// ---- VISUs/Keypad.TcVIS
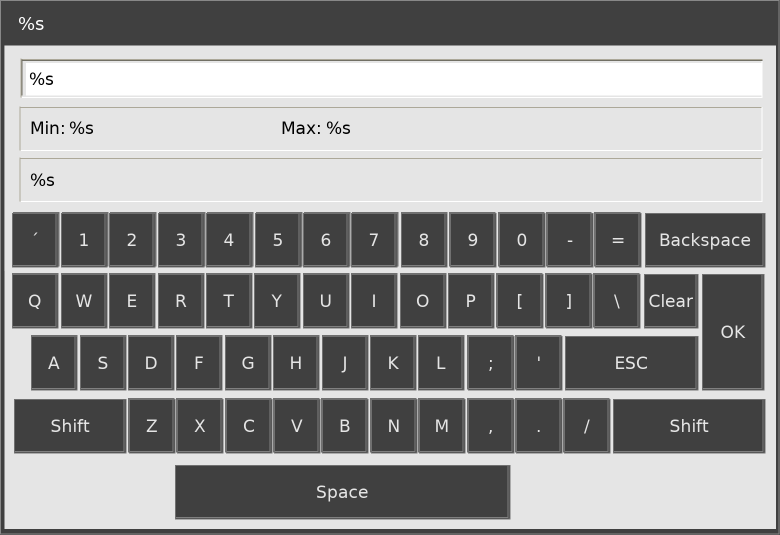
VISUALIZATION Keypad  // 780x535
VAR_INPUT
	stVariableValue : STRING;
	stMin : STRING;
	stMax : STRING;
	stTitle : STRING;
	flags : DWORD;
END_VAR
VAR
	bInit : BOOL;
	bShift : BOOL;
	stMessage : STRING;
	stOutputValue : STRING;
END_VAR
    Rectangle (5,201 772x70)
    Rectangle (3,271 775x62)
    Rectangle (3,333 775x63)
    Rectangle (3,396 775x62)
    Rectangle (3,455 775x75)
    Button (702,274 62x116), "OK"
        OnMouseDown: CloseDialog Dialog=Keypad, Result=OK, NumpadKeypad=True, NumpadKeypadSet=True
    Button (565,336 133x54), "ESC"
        OnMouseDown: CloseDialog Dialog=Keypad, Result=Cancel, NumpadKeypad=True, NumpadKeypadSet=True
    Button (644,274 54x54), "Clear"
        OnMouseDown: execute { stVariableValue := ''; stOutputValue := ''; }
    Button (645,213 120x54), "Backspace"
        OnMouseDown: execute { VisuDlg_CheckedBack(stOutputValue, stVariableValue, bInit); }
    Button (613,399 152x54), "Shift"
        OnMouseDown: toggle bShift
    Button (175,465 335x54), "Space"
        OnMouseDown: execute { VisuDlg_CheckedAppend(stOutputValue, stVariableValue, bInit, (flags AND VisuElems.Visu_InputFlags.Password) = 1, ' '); }
    Button (593,273 46x54), "|", invisible if: NOT bShift
        OnMouseDown: execute { VisuDlg_CheckedAppend(stOutputValue, stVariableValue, bInit, (flags AND VisuElems.Visu_InputFlags.Password) = 1, '|'); }
    Button (467,398 46x54), "<", invisible if: NOT bShift
        OnMouseDown: execute { VisuDlg_CheckedAppend(stOutputValue, stVariableValue, bInit, (flags AND VisuElems.Visu_InputFlags.Password) = 1, '<'); }
    Button (515,398 46x54), ">", invisible if: NOT bShift
        OnMouseDown: execute { VisuDlg_CheckedAppend(stOutputValue, stVariableValue, bInit, (flags AND VisuElems.Visu_InputFlags.Password) = 1, '>'); }
    Button (254,273 46x54), "y", invisible if: NOT bShift
        OnMouseDown: execute { VisuDlg_CheckedAppend(stOutputValue, stVariableValue, bInit, (flags AND VisuElems.Visu_InputFlags.Password) = 1, 'y'); }
    Button (254,274 46x54), "Y", invisible if: bShift
        OnMouseDown: execute { VisuDlg_CheckedAppend(stOutputValue, stVariableValue, bInit, (flags AND VisuElems.Visu_InputFlags.Password) = 1, 'Y'); }
    Button (176,398 46x54), "x", invisible if: NOT bShift
        OnMouseDown: execute { VisuDlg_CheckedAppend(stOutputValue, stVariableValue, bInit, (flags AND VisuElems.Visu_InputFlags.Password) = 1, 'x'); }
    Button (177,399 46x54), "X", invisible if: bShift
        OnMouseDown: execute { VisuDlg_CheckedAppend(stOutputValue, stVariableValue, bInit, (flags AND VisuElems.Visu_InputFlags.Password) = 1, 'X'); }
    Button (225,398 46x54), "c", invisible if: NOT bShift
        OnMouseDown: execute { VisuDlg_CheckedAppend(stOutputValue, stVariableValue, bInit, (flags AND VisuElems.Visu_InputFlags.Password) = 1, 'c'); }
    Button (226,399 46x54), "C", invisible if: bShift
        OnMouseDown: execute { VisuDlg_CheckedAppend(stOutputValue, stVariableValue, bInit, (flags AND VisuElems.Visu_InputFlags.Password) = 1, 'C'); }
    Button (273,398 46x54), "v", invisible if: NOT bShift
        OnMouseDown: execute { VisuDlg_CheckedAppend(stOutputValue, stVariableValue, bInit, (flags AND VisuElems.Visu_InputFlags.Password) = 1, 'v'); }
    Button (274,399 46x54), "V", invisible if: bShift
        OnMouseDown: execute { VisuDlg_CheckedAppend(stOutputValue, stVariableValue, bInit, (flags AND VisuElems.Visu_InputFlags.Password) = 1, 'V'); }
    Button (321,398 46x54), "b", invisible if: NOT bShift
        OnMouseDown: execute { VisuDlg_CheckedAppend(stOutputValue, stVariableValue, bInit, (flags AND VisuElems.Visu_InputFlags.Password) = 1, 'b'); }
    Button (322,399 46x54), "B", invisible if: bShift
        OnMouseDown: execute { VisuDlg_CheckedAppend(stOutputValue, stVariableValue, bInit, (flags AND VisuElems.Visu_InputFlags.Password) = 1, 'B'); }
    Button (370,398 46x54), "n", invisible if: NOT bShift
        OnMouseDown: execute { VisuDlg_CheckedAppend(stOutputValue, stVariableValue, bInit, (flags AND VisuElems.Visu_InputFlags.Password) = 1, 'n'); }
    Button (371,399 46x54), "N", invisible if: bShift
        OnMouseDown: execute { VisuDlg_CheckedAppend(stOutputValue, stVariableValue, bInit, (flags AND VisuElems.Visu_InputFlags.Password) = 1, 'N'); }
    Button (418,398 46x54), "m", invisible if: NOT bShift
        OnMouseDown: execute { VisuDlg_CheckedAppend(stOutputValue, stVariableValue, bInit, (flags AND VisuElems.Visu_InputFlags.Password) = 1, 'm'); }
    Button (419,399 46x54), "M", invisible if: bShift
        OnMouseDown: execute { VisuDlg_CheckedAppend(stOutputValue, stVariableValue, bInit, (flags AND VisuElems.Visu_InputFlags.Password) = 1, 'M'); }
    Button (467,335 46x54), ":", invisible if: NOT bShift
        OnMouseDown: execute { VisuDlg_CheckedAppend(stOutputValue, stVariableValue, bInit, (flags AND VisuElems.Visu_InputFlags.Password) = 1, ':'); }
    Button (546,212 45x54), "_", invisible if: NOT bShift
        OnMouseDown: execute { VisuDlg_CheckedAppend(stOutputValue, stVariableValue, bInit, (flags AND VisuElems.Visu_InputFlags.Password) = 1, '_'); }
    Button (31,335 46x54), "a", invisible if: NOT bShift
        OnMouseDown: execute { VisuDlg_CheckedAppend(stOutputValue, stVariableValue, bInit, (flags AND VisuElems.Visu_InputFlags.Password) = 1, 'a'); }
    Button (31,336 46x54), "A", invisible if: bShift
        OnMouseDown: execute { VisuDlg_CheckedAppend(stOutputValue, stVariableValue, bInit, (flags AND VisuElems.Visu_InputFlags.Password) = 1, 'A'); }
    Button (80,335 46x54), "s", invisible if: NOT bShift
        OnMouseDown: execute { VisuDlg_CheckedAppend(stOutputValue, stVariableValue, bInit, (flags AND VisuElems.Visu_InputFlags.Password) = 1, 's'); }
    Button (80,336 46x54), "S", invisible if: bShift
        OnMouseDown: execute { VisuDlg_CheckedAppend(stOutputValue, stVariableValue, bInit, (flags AND VisuElems.Visu_InputFlags.Password) = 1, 'S'); }
    Button (128,335 46x54), "d", invisible if: NOT bShift
        OnMouseDown: execute { VisuDlg_CheckedAppend(stOutputValue, stVariableValue, bInit, (flags AND VisuElems.Visu_InputFlags.Password) = 1, 'd'); }
    Button (128,336 46x54), "D", invisible if: bShift
        OnMouseDown: execute { VisuDlg_CheckedAppend(stOutputValue, stVariableValue, bInit, (flags AND VisuElems.Visu_InputFlags.Password) = 1, 'D'); }
    Button (176,335 46x54), "f", invisible if: NOT bShift
        OnMouseDown: execute { VisuDlg_CheckedAppend(stOutputValue, stVariableValue, bInit, (flags AND VisuElems.Visu_InputFlags.Password) = 1, 'f'); }
    Button (176,336 46x54), "F", invisible if: bShift
        OnMouseDown: execute { VisuDlg_CheckedAppend(stOutputValue, stVariableValue, bInit, (flags AND VisuElems.Visu_InputFlags.Password) = 1, 'F'); }
    Button (225,335 46x54), "g", invisible if: NOT bShift
        OnMouseDown: execute { VisuDlg_CheckedAppend(stOutputValue, stVariableValue, bInit, (flags AND VisuElems.Visu_InputFlags.Password) = 1, 'g'); }
    Button (225,336 46x54), "G", invisible if: bShift
        OnMouseDown: execute { VisuDlg_CheckedAppend(stOutputValue, stVariableValue, bInit, (flags AND VisuElems.Visu_InputFlags.Password) = 1, 'G'); }
    Button (273,335 46x54), "h", invisible if: NOT bShift
        OnMouseDown: execute { VisuDlg_CheckedAppend(stOutputValue, stVariableValue, bInit, (flags AND VisuElems.Visu_InputFlags.Password) = 1, 'h'); }
    Button (273,336 46x54), "H", invisible if: bShift
        OnMouseDown: execute { VisuDlg_CheckedAppend(stOutputValue, stVariableValue, bInit, (flags AND VisuElems.Visu_InputFlags.Password) = 1, 'H'); }
    Button (322,335 46x54), "j", invisible if: NOT bShift
        OnMouseDown: execute { VisuDlg_CheckedAppend(stOutputValue, stVariableValue, bInit, (flags AND VisuElems.Visu_InputFlags.Password) = 1, 'j'); }
    Button (322,336 46x54), "J", invisible if: bShift
        OnMouseDown: execute { VisuDlg_CheckedAppend(stOutputValue, stVariableValue, bInit, (flags AND VisuElems.Visu_InputFlags.Password) = 1, 'J'); }
    Button (370,335 46x54), "k", invisible if: NOT bShift
        OnMouseDown: execute { VisuDlg_CheckedAppend(stOutputValue, stVariableValue, bInit, (flags AND VisuElems.Visu_InputFlags.Password) = 1, 'k'); }
    Button (370,336 46x54), "K", invisible if: bShift
        OnMouseDown: execute { VisuDlg_CheckedAppend(stOutputValue, stVariableValue, bInit, (flags AND VisuElems.Visu_InputFlags.Password) = 1, 'K'); }
    Button (418,335 46x54), "l", invisible if: NOT bShift
        OnMouseDown: execute { VisuDlg_CheckedAppend(stOutputValue, stVariableValue, bInit, (flags AND VisuElems.Visu_InputFlags.Password) = 1, 'l'); }
    Button (418,336 46x54), "L", invisible if: bShift
        OnMouseDown: execute { VisuDlg_CheckedAppend(stOutputValue, stVariableValue, bInit, (flags AND VisuElems.Visu_InputFlags.Password) = 1, 'L'); }
    Button (159,212 46x54), "#", invisible if: NOT bShift
        OnMouseDown: execute { VisuDlg_CheckedAppend(stOutputValue, stVariableValue, bInit, (flags AND VisuElems.Visu_InputFlags.Password) = 1, '#'); }
    Button (110,212 46x54), "@", invisible if: NOT bShift
        OnMouseDown: execute { VisuDlg_CheckedAppend(stOutputValue, stVariableValue, bInit, (flags AND VisuElems.Visu_InputFlags.Password) = 1, '@'); }
    Button (12,273 46x54), "q", invisible if: NOT bShift
        OnMouseDown: execute { VisuDlg_CheckedAppend(stOutputValue, stVariableValue, bInit, (flags AND VisuElems.Visu_InputFlags.Password) = 1, 'q'); }
    Button (12,274 46x54), "Q", invisible if: bShift
        OnMouseDown: execute { VisuDlg_CheckedAppend(stOutputValue, stVariableValue, bInit, (flags AND VisuElems.Visu_InputFlags.Password) = 1, 'Q'); }
    Button (61,273 46x54), "w", invisible if: NOT bShift
        OnMouseDown: execute { VisuDlg_CheckedAppend(stOutputValue, stVariableValue, bInit, (flags AND VisuElems.Visu_InputFlags.Password) = 1, 'w'); }
    Button (61,274 46x54), "W", invisible if: bShift
        OnMouseDown: execute { VisuDlg_CheckedAppend(stOutputValue, stVariableValue, bInit, (flags AND VisuElems.Visu_InputFlags.Password) = 1, 'W'); }
    Button (109,273 46x54), "e", invisible if: NOT bShift
        OnMouseDown: execute { VisuDlg_CheckedAppend(stOutputValue, stVariableValue, bInit, (flags AND VisuElems.Visu_InputFlags.Password) = 1, 'e'); }
    Button (109,274 46x54), "E", invisible if: bShift
        OnMouseDown: execute { VisuDlg_CheckedAppend(stOutputValue, stVariableValue, bInit, (flags AND VisuElems.Visu_InputFlags.Password) = 1, 'E'); }
    Button (158,273 46x54), "r", invisible if: NOT bShift
        OnMouseDown: execute { VisuDlg_CheckedAppend(stOutputValue, stVariableValue, bInit, (flags AND VisuElems.Visu_InputFlags.Password) = 1, 'r'); }
    Button (158,274 46x54), "R", invisible if: bShift
        OnMouseDown: execute { VisuDlg_CheckedAppend(stOutputValue, stVariableValue, bInit, (flags AND VisuElems.Visu_InputFlags.Password) = 1, 'R'); }
    Button (206,273 46x54), "t", invisible if: NOT bShift
        OnMouseDown: execute { VisuDlg_CheckedAppend(stOutputValue, stVariableValue, bInit, (flags AND VisuElems.Visu_InputFlags.Password) = 1, 't'); }
    Button (206,274 46x54), "T", invisible if: bShift
        OnMouseDown: execute { VisuDlg_CheckedAppend(stOutputValue, stVariableValue, bInit, (flags AND VisuElems.Visu_InputFlags.Password) = 1, 'T'); }
    Button (128,398 46x54), "z", invisible if: NOT bShift
        OnMouseDown: execute { VisuDlg_CheckedAppend(stOutputValue, stVariableValue, bInit, (flags AND VisuElems.Visu_InputFlags.Password) = 1, 'z'); }
    Button (129,399 46x54), "Z", invisible if: bShift
        OnMouseDown: execute { VisuDlg_CheckedAppend(stOutputValue, stVariableValue, bInit, (flags AND VisuElems.Visu_InputFlags.Password) = 1, 'Z'); }
    Button (303,273 46x54), "u", invisible if: NOT bShift
        OnMouseDown: execute { VisuDlg_CheckedAppend(stOutputValue, stVariableValue, bInit, (flags AND VisuElems.Visu_InputFlags.Password) = 1, 'u'); }
    Button (303,274 46x54), "U", invisible if: bShift
        OnMouseDown: execute { VisuDlg_CheckedAppend(stOutputValue, stVariableValue, bInit, (flags AND VisuElems.Visu_InputFlags.Password) = 1, 'U'); }
    Button (351,273 46x54), "i", invisible if: NOT bShift
        OnMouseDown: execute { VisuDlg_CheckedAppend(stOutputValue, stVariableValue, bInit, (flags AND VisuElems.Visu_InputFlags.Password) = 1, 'i'); }
    Button (351,274 46x54), "I", invisible if: bShift
        OnMouseDown: execute { VisuDlg_CheckedAppend(stOutputValue, stVariableValue, bInit, (flags AND VisuElems.Visu_InputFlags.Password) = 1, 'I'); }
    Button (400,273 46x54), "o", invisible if: NOT bShift
        OnMouseDown: execute { VisuDlg_CheckedAppend(stOutputValue, stVariableValue, bInit, (flags AND VisuElems.Visu_InputFlags.Password) = 1, 'o'); }
    Button (400,274 46x54), "O", invisible if: bShift
        OnMouseDown: execute { VisuDlg_CheckedAppend(stOutputValue, stVariableValue, bInit, (flags AND VisuElems.Visu_InputFlags.Password) = 1, 'O'); }
    Button (448,273 46x54), "p", invisible if: NOT bShift
        OnMouseDown: execute { VisuDlg_CheckedAppend(stOutputValue, stVariableValue, bInit, (flags AND VisuElems.Visu_InputFlags.Password) = 1, 'p'); }
    Button (448,274 46x54), "P", invisible if: bShift
        OnMouseDown: execute { VisuDlg_CheckedAppend(stOutputValue, stVariableValue, bInit, (flags AND VisuElems.Visu_InputFlags.Password) = 1, 'P'); }
    Button (594,212 46x54), "+", invisible if: NOT bShift
        OnMouseDown: execute { VisuDlg_CheckedAppend(stOutputValue, stVariableValue, bInit, (flags AND VisuElems.Visu_InputFlags.Password) = 1, '+'); }
    Button (401,212 46x54), "*", invisible if: NOT bShift
        OnMouseDown: execute { VisuDlg_CheckedAppend(stOutputValue, stVariableValue, bInit, (flags AND VisuElems.Visu_InputFlags.Password) = 1, '*'); }
    Button (13,212 46x54), "~", invisible if: NOT bShift
        OnMouseDown: execute { VisuDlg_CheckedAppend(stOutputValue, stVariableValue, bInit, (flags AND VisuElems.Visu_InputFlags.Password) = 1, '~'); }
    Button (304,212 46x54), "^", invisible if: NOT bShift
        OnMouseDown: execute { VisuDlg_CheckedAppend(stOutputValue, stVariableValue, bInit, (flags AND VisuElems.Visu_InputFlags.Password) = 1, '^'); }
    Button (62,212 46x54), "!", invisible if: NOT bShift
        OnMouseDown: execute { VisuDlg_CheckedAppend(stOutputValue, stVariableValue, bInit, (flags AND VisuElems.Visu_InputFlags.Password) = 1, '!'); }
    Button (515,335 46x54), """, invisible if: NOT bShift
        OnMouseDown: execute { VisuDlg_CheckedAppend(stOutputValue, stVariableValue, bInit, (flags AND VisuElems.Visu_InputFlags.Password) = 1, '"'); }
    Button (207,212 46x54), "$", invisible if: NOT bShift
        OnMouseDown: execute { VisuDlg_CheckedAppend(stOutputValue, stVariableValue, bInit, (flags AND VisuElems.Visu_InputFlags.Password) = 1, '$$'); }
    Button (256,212 46x54), "%", invisible if: NOT bShift
        OnMouseDown: execute { VisuDlg_CheckedAppend(stOutputValue, stVariableValue, bInit, (flags AND VisuElems.Visu_InputFlags.Password) = 1, '%'); }
    Button (352,212 46x54), "&", invisible if: NOT bShift
        OnMouseDown: execute { VisuDlg_CheckedAppend(stOutputValue, stVariableValue, bInit, (flags AND VisuElems.Visu_InputFlags.Password) = 1, '&'); }
    Button (449,212 46x54), "(", invisible if: NOT bShift
        OnMouseDown: execute { VisuDlg_CheckedAppend(stOutputValue, stVariableValue, bInit, (flags AND VisuElems.Visu_InputFlags.Password) = 1, '('); }
    Button (498,212 46x54), ")", invisible if: NOT bShift
        OnMouseDown: execute { VisuDlg_CheckedAppend(stOutputValue, stVariableValue, bInit, (flags AND VisuElems.Visu_InputFlags.Password) = 1, ')'); }
    Button (563,398 46x54), "?", invisible if: NOT bShift
        OnMouseDown: execute { VisuDlg_CheckedAppend(stOutputValue, stVariableValue, bInit, (flags AND VisuElems.Visu_InputFlags.Password) = 1, '?'); }
    Rectangle (5,104 773x97)
    Rectangle (27,164 734x32), "%s", text variable: stMessage
    Rectangle (5,42 773x62)
    Rectangle (776,0 4x530)
    Rectangle (0,2 4x527)
    Rectangle (0,529 780x6)
    Polyline (20,201) (20,158) (762,158)
    Polyline (20,150) (20,107) (762,107)
    Polyline (21,97) (21,59) (762,59)
    Polyline (21,201) (762,201) (762,158)
    Polyline (21,150) (762,150) (762,107)
    Polyline (22,97) (762,97) (762,60)
    Rectangle (0,0 779x45)
    Rectangle (15,8 757x32), "%s", text variable: stTitle
    Polyline (22,95) (22,60) (762,60)
    Rectangle (26,63 736x32), "%s", text variable: stOutputValue
    Rectangle (27,112 42x32), "Min:", text variable: stMin, invisible if: LEN(stMin) = 0
    Rectangle (66,112 157x32), "%s", text variable: stMin, invisible if: LEN(stMin) = 0
    Rectangle (278,112 45x32), "Max:", text variable: stMin, invisible if: LEN(stMax) = 0
    Rectangle (323,112 217x32), "%s", text variable: stMax, invisible if: LEN(stMax) = 0
    Button (12,213 46x54), "´", invisible if: bShift
        OnMouseDown: execute { VisuDlg_CheckedAppend(stOutputValue, stVariableValue, bInit, (flags AND VisuElems.Visu_InputFlags.Password) = 1, '´'); }
    Button (61,213 46x54), "1", invisible if: bShift
        OnMouseDown: execute { VisuDlg_CheckedAppend(stOutputValue, stVariableValue, bInit, (flags AND VisuElems.Visu_InputFlags.Password) = 1, '1'); }
    Button (109,213 46x54), "2", invisible if: bShift
        OnMouseDown: execute { VisuDlg_CheckedAppend(stOutputValue, stVariableValue, bInit, (flags AND VisuElems.Visu_InputFlags.Password) = 1, '2'); }
    Button (158,213 46x54), "3", invisible if: bShift
        OnMouseDown: execute { VisuDlg_CheckedAppend(stOutputValue, stVariableValue, bInit, (flags AND VisuElems.Visu_InputFlags.Password) = 1, '3'); }
    Button (206,213 46x54), "4", invisible if: bShift
        OnMouseDown: execute { VisuDlg_CheckedAppend(stOutputValue, stVariableValue, bInit, (flags AND VisuElems.Visu_InputFlags.Password) = 1, '4'); }
    Button (255,213 46x54), "5", invisible if: bShift
        OnMouseDown: execute { VisuDlg_CheckedAppend(stOutputValue, stVariableValue, bInit, (flags AND VisuElems.Visu_InputFlags.Password) = 1, '5'); }
    Button (303,213 46x54), "6", invisible if: bShift
        OnMouseDown: execute { VisuDlg_CheckedAppend(stOutputValue, stVariableValue, bInit, (flags AND VisuElems.Visu_InputFlags.Password) = 1, '6'); }
    Button (351,213 46x54), "7", invisible if: bShift
        OnMouseDown: execute { VisuDlg_CheckedAppend(stOutputValue, stVariableValue, bInit, (flags AND VisuElems.Visu_InputFlags.Password) = 1, '7'); }
    Button (401,213 46x54), "8", invisible if: bShift
        OnMouseDown: execute { VisuDlg_CheckedAppend(stOutputValue, stVariableValue, bInit, (flags AND VisuElems.Visu_InputFlags.Password) = 1, '8'); }
    Button (450,213 46x54), "9", invisible if: bShift
        OnMouseDown: execute { VisuDlg_CheckedAppend(stOutputValue, stVariableValue, bInit, (flags AND VisuElems.Visu_InputFlags.Password) = 1, '9'); }
    Button (499,213 46x54), "0", invisible if: bShift
        OnMouseDown: execute { VisuDlg_CheckedAppend(stOutputValue, stVariableValue, bInit, (flags AND VisuElems.Visu_InputFlags.Password) = 1, '0'); }
    Button (547,213 46x54), "-", invisible if: bShift
        OnMouseDown: execute { VisuDlg_CheckedAppend(stOutputValue, stVariableValue, bInit, (flags AND VisuElems.Visu_InputFlags.Password) = 1, '-'); }
    Button (595,213 46x54), "=", invisible if: bShift
        OnMouseDown: execute { VisuDlg_CheckedAppend(stOutputValue, stVariableValue, bInit, (flags AND VisuElems.Visu_InputFlags.Password) = 1, '='); }
    Button (496,273 46x54), "{", invisible if: NOT bShift
        OnMouseDown: execute { VisuDlg_CheckedAppend(stOutputValue, stVariableValue, bInit, (flags AND VisuElems.Visu_InputFlags.Password) = 1, '{'); }
    Button (497,274 46x54), "[", invisible if: bShift
        OnMouseDown: execute { VisuDlg_CheckedAppend(stOutputValue, stVariableValue, bInit, (flags AND VisuElems.Visu_InputFlags.Password) = 1, '['); }
    Button (545,273 46x54), "}", invisible if: NOT bShift
        OnMouseDown: execute { VisuDlg_CheckedAppend(stOutputValue, stVariableValue, bInit, (flags AND VisuElems.Visu_InputFlags.Password) = 1, '}'); }
    Button (546,274 46x54), "]", invisible if: bShift
        OnMouseDown: execute { VisuDlg_CheckedAppend(stOutputValue, stVariableValue, bInit, (flags AND VisuElems.Visu_InputFlags.Password) = 1, ']'); }
    Button (594,274 46x54), "\", invisible if: bShift
        OnMouseDown: execute { VisuDlg_CheckedAppend(stOutputValue, stVariableValue, bInit, (flags AND VisuElems.Visu_InputFlags.Password) = 1, '\'); }
    Button (468,336 46x54), ";", invisible if: bShift
        OnMouseDown: execute { VisuDlg_CheckedAppend(stOutputValue, stVariableValue, bInit, (flags AND VisuElems.Visu_InputFlags.Password) = 1, ';'); }
    Button (516,336 46x54), "'", invisible if: bShift
        OnMouseDown: execute { VisuDlg_CheckedAppend(stOutputValue, stVariableValue, bInit, (flags AND VisuElems.Visu_InputFlags.Password) = 1, '$''); }
    Button (468,399 46x54), ",", invisible if: bShift
        OnMouseDown: execute { VisuDlg_CheckedAppend(stOutputValue, stVariableValue, bInit, (flags AND VisuElems.Visu_InputFlags.Password) = 1, ','); }
    Button (516,399 46x54), ".", invisible if: bShift
        OnMouseDown: execute { VisuDlg_CheckedAppend(stOutputValue, stVariableValue, bInit, (flags AND VisuElems.Visu_InputFlags.Password) = 1, '.'); }
    Button (564,399 46x54), "/", invisible if: bShift
        OnMouseDown: execute { VisuDlg_CheckedAppend(stOutputValue, stVariableValue, bInit, (flags AND VisuElems.Visu_InputFlags.Password) = 1, '/'); }
    Button (14,399 112x54), "Shift"
        OnMouseDown: toggle bShift
    hotkey HotkeyInput Id=481083523072, Key=KeyDown=True, KeyName=BACKSPACE, ActionToExecute=Action=STSnippet=VisuDlg_CheckedBack(stOutputValue, stVariableValue, bInit);, VisuElemId=-1
    hotkey HotkeyInput Id=481084571648, Key=KeyDown=True, KeyName=DELETE, ActionToExecute=Action=STSnippet=stVariableValue := ''; stOutputValue := '';, VisuElemId=-1
    hotkey HotkeyInput Id=481085620224, Key=KeyDown=True, KeyName=ESCAPE, ActionToExecute=Action=Dialog=Keypad, Result=Cancel, NumpadKeypad=True, NumpadKeypadSet=True, VisuElemId=-1
    hotkey HotkeyInput Id=481086668800, Key=KeyDown=True, KeyName=SPACE, ActionToExecute=Action=STSnippet=VisuDlg_CheckedAppend(stOutputValue, stVariableValue, bInit, (flags AND VisuElems.Visu_InputFlags.Password) = 1, ' ');, VisuElemId=-1
    hotkey HotkeyInput Id=481087717376, Key=Modifiers=1, KeyDown=True, KeyName=SPACE, ActionToExecute=Action=ToggleVariable=bShift, VisuElemId=-1
    hotkey HotkeyInput Id=481088765952, Key=KeyDown=True, KeyName=RETURN_KEY, ActionToExecute=Action=Dialog=Keypad, Result=OK, NumpadKeypad=True, NumpadKeypadSet=True, VisuElemId=-1
    hotkey HotkeyInput Id=481089814528, Key=KeyDown=True, KeyName=1, ActionToExecute=Action=STSnippet=IF bShift THEN VisuDlg_CheckedAppend(stOutputValue, stVariableValue, bInit, (flags AND VisuElems.Visu_InputFlags.Password) = 1, '!'); ELSE VisuDlg_CheckedAppend(stOutputValue, stVariableValue, bInit, (flags AND VisuElems.Visu_InputFlags.Password) = 1, '1'); END_IF, VisuElemId=-1
    hotkey HotkeyInput Id=481090863104, Key=KeyDown=True, KeyName=2, ActionToExecute=Action=STSnippet=IF bShift THEN VisuDlg_CheckedAppend(stOutputValue, stVariableValue, bInit, (flags AND VisuElems.Visu_InputFlags.Password) = 1, '@'); ELSE VisuDlg_CheckedAppend(stOutputValue, stVariableValue, bInit, (flags AND VisuElems.Visu_InputFlags.Password) = 1, '2'); END_IF, VisuElemId=-1
    hotkey HotkeyInput Id=481091911680, Key=KeyDown=True, KeyName=3, ActionToExecute=Action=STSnippet=IF bShift THEN VisuDlg_CheckedAppend(stOutputValue, stVariableValue, bInit, (flags AND VisuElems.Visu_InputFlags.Password) = 1, '#'); ELSE VisuDlg_CheckedAppend(stOutputValue, stVariableValue, bInit, (flags AND VisuElems.Visu_InputFlags.Password) = 1, '3'); END_IF, VisuElemId=-1
    hotkey HotkeyInput Id=481092960256, Key=KeyDown=True, KeyName=4, ActionToExecute=Action=STSnippet=IF bShift THEN VisuDlg_CheckedAppend(stOutputValue, stVariableValue, bInit, (flags AND VisuElems.Visu_InputFlags.Password) = 1, '$$'); ELSE VisuDlg_CheckedAppend(stOutputValue, stVariableValue, bInit, (flags AND VisuElems.Visu_InputFlags.Password) = 1, '4'); END_IF, VisuElemId=-1
    hotkey HotkeyInput Id=481094008832, Key=KeyDown=True, KeyName=5, ActionToExecute=Action=STSnippet=IF bShift THEN VisuDlg_CheckedAppend(stOutputValue, stVariableValue, bInit, (flags AND VisuElems.Visu_InputFlags.Password) = 1, '%'); ELSE VisuDlg_CheckedAppend(stOutputValue, stVariableValue, bInit, (flags AND VisuElems.Visu_InputFlags.Password) = 1, '5'); END_IF, VisuElemId=-1
    hotkey HotkeyInput Id=481095057408, Key=KeyDown=True, KeyName=6, ActionToExecute=Action=STSnippet=IF bShift THEN VisuDlg_CheckedAppend(stOutputValue, stVariableValue, bInit, (flags AND VisuElems.Visu_InputFlags.Password) = 1, '^'); ELSE VisuDlg_CheckedAppend(stOutputValue, stVariableValue, bInit, (flags AND VisuElems.Visu_InputFlags.Password) = 1, '6'); END_IF, VisuElemId=-1
    hotkey HotkeyInput Id=481096105984, Key=KeyDown=True, KeyName=7, ActionToExecute=Action=STSnippet=IF bShift THEN VisuDlg_CheckedAppend(stOutputValue, stVariableValue, bInit, (flags AND VisuElems.Visu_InputFlags.Password) = 1, '&'); ELSE VisuDlg_CheckedAppend(stOutputValue, stVariableValue, bInit, (flags AND VisuElems.Visu_InputFlags.Password) = 1, '7'); END_IF, VisuElemId=-1
    hotkey HotkeyInput Id=481097154560, Key=KeyDown=True, KeyName=8, ActionToExecute=Action=STSnippet=IF bShift THEN VisuDlg_CheckedAppend(stOutputValue, stVariableValue, bInit, (flags AND VisuElems.Visu_InputFlags.Password) = 1, '*'); ELSE VisuDlg_CheckedAppend(stOutputValue, stVariableValue, bInit, (flags AND VisuElems.Visu_InputFlags.Password) = 1, '8'); END_IF, VisuElemId=-1
    hotkey HotkeyInput Id=481098203136, Key=KeyDown=True, KeyName=9, ActionToExecute=Action=STSnippet=IF bShift THEN VisuDlg_CheckedAppend(stOutputValue, stVariableValue, bInit, (flags AND VisuElems.Visu_InputFlags.Password) = 1, '('); ELSE VisuDlg_CheckedAppend(stOutputValue, stVariableValue, bInit, (flags AND VisuElems.Visu_InputFlags.Password) = 1, '9'); END_IF, VisuElemId=-1
    hotkey HotkeyInput Id=481099251712, Key=KeyDown=True, KeyName=0, ActionToExecute=Action=STSnippet=IF bShift THEN VisuDlg_CheckedAppend(stOutputValue, stVariableValue, bInit, (flags AND VisuElems.Visu_InputFlags.Password) = 1, ')'); ELSE VisuDlg_CheckedAppend(stOutputValue, stVariableValue, bInit, (flags AND VisuElems.Visu_InputFlags.Password) = 1, '0'); END_IF, VisuElemId=-1
    hotkey HotkeyInput Id=481100300288, Key=KeyDown=True, KeyName=SUBTRACT, ActionToExecute=Action=STSnippet=IF bShift THEN VisuDlg_CheckedAppend(stOutputValue, stVariableValue, bInit, (flags AND VisuElems.Visu_InputFlags.Password) = 1, '_'); ELSE VisuDlg_CheckedAppend(stOutputValue, stVariableValue, bInit, (flags AND VisuElems.Visu_InputFlags.Password) = 1, '-'); END_IF, VisuElemId=-1
    hotkey HotkeyInput Id=481101348864, Key=KeyDown=True, KeyName=ADDITION, ActionToExecute=Action=STSnippet=IF bShift THEN VisuDlg_CheckedAppend(stOutputValue, stVariableValue, bInit, (flags AND VisuElems.Visu_InputFlags.Password) = 1, '='); ELSE VisuDlg_CheckedAppend(stOutputValue, stVariableValue, bInit, (flags AND VisuElems.Visu_InputFlags.Password) = 1, '+'); END_IF, VisuElemId=-1
    hotkey HotkeyInput Id=481102397440, Key=KeyDown=True, KeyName=Q, ActionToExecute=Action=STSnippet=IF bShift THEN VisuDlg_CheckedAppend(stOutputValue, stVariableValue, bInit, (flags AND VisuElems.Visu_InputFlags.Password) = 1, 'q'); ELSE VisuDlg_CheckedAppend(stOutputValue, stVariableValue, bInit, (flags AND VisuElems.Visu_InputFlags.Password) = 1, 'Q'); END_IF, VisuElemId=-1
    hotkey HotkeyInput Id=481103446016, Key=KeyDown=True, KeyName=W, ActionToExecute=Action=STSnippet=IF bShift THEN VisuDlg_CheckedAppend(stOutputValue, stVariableValue, bInit, (flags AND VisuElems.Visu_InputFlags.Password) = 1, 'w'); ELSE VisuDlg_CheckedAppend(stOutputValue, stVariableValue, bInit, (flags AND VisuElems.Visu_InputFlags.Password) = 1, 'W'); END_IF, VisuElemId=-1
    hotkey HotkeyInput Id=481104494592, Key=KeyDown=True, KeyName=E, ActionToExecute=Action=STSnippet=IF bShift THEN VisuDlg_CheckedAppend(stOutputValue, stVariableValue, bInit, (flags AND VisuElems.Visu_InputFlags.Password) = 1, 'e'); ELSE VisuDlg_CheckedAppend(stOutputValue, stVariableValue, bInit, (flags AND VisuElems.Visu_InputFlags.Password) = 1, 'E'); END_IF, VisuElemId=-1
    hotkey HotkeyInput Id=481105543168, Key=KeyDown=True, KeyName=R, ActionToExecute=Action=STSnippet=IF bShift THEN VisuDlg_CheckedAppend(stOutputValue, stVariableValue, bInit, (flags AND VisuElems.Visu_InputFlags.Password) = 1, 'r'); ELSE VisuDlg_CheckedAppend(stOutputValue, stVariableValue, bInit, (flags AND VisuElems.Visu_InputFlags.Password) = 1, 'R'); END_IF, VisuElemId=-1
    hotkey HotkeyInput Id=481106591744, Key=KeyDown=True, KeyName=T, ActionToExecute=Action=STSnippet=IF bShift THEN VisuDlg_CheckedAppend(stOutputValue, stVariableValue, bInit, (flags AND VisuElems.Visu_InputFlags.Password) = 1, 't'); ELSE VisuDlg_CheckedAppend(stOutputValue, stVariableValue, bInit, (flags AND VisuElems.Visu_InputFlags.Password) = 1, 'T'); END_IF, VisuElemId=-1
    hotkey HotkeyInput Id=481107640320, Key=KeyDown=True, KeyName=Y, ActionToExecute=Action=STSnippet=IF bShift THEN VisuDlg_CheckedAppend(stOutputValue, stVariableValue, bInit, (flags AND VisuElems.Visu_InputFlags.Password) = 1, 'y'); ELSE VisuDlg_CheckedAppend(stOutputValue, stVariableValue, bInit, (flags AND VisuElems.Visu_InputFlags.Password) = 1, 'Y'); END_IF, VisuElemId=-1
    hotkey HotkeyInput Id=481108688896, Key=KeyDown=True, KeyName=U, ActionToExecute=Action=STSnippet=IF bShift THEN VisuDlg_CheckedAppend(stOutputValue, stVariableValue, bInit, (flags AND VisuElems.Visu_InputFlags.Password) = 1, 'u'); ELSE VisuDlg_CheckedAppend(stOutputValue, stVariableValue, bInit, (flags AND VisuElems.Visu_InputFlags.Password) = 1, 'U'); END_IF, VisuElemId=-1
    hotkey HotkeyInput Id=481109737472, Key=KeyDown=True, KeyName=I, ActionToExecute=Action=STSnippet=IF bShift THEN VisuDlg_CheckedAppend(stOutputValue, stVariableValue, bInit, (flags AND VisuElems.Visu_InputFlags.Password) = 1, 'i'); ELSE VisuDlg_CheckedAppend(stOutputValue, stVariableValue, bInit, (flags AND VisuElems.Visu_InputFlags.Password) = 1, 'I'); END_IF, VisuElemId=-1
    hotkey HotkeyInput Id=481110786048, Key=KeyDown=True, KeyName=O, ActionToExecute=Action=STSnippet=IF bShift THEN VisuDlg_CheckedAppend(stOutputValue, stVariableValue, bInit, (flags AND VisuElems.Visu_InputFlags.Password) = 1, 'o'); ELSE VisuDlg_CheckedAppend(stOutputValue, stVariableValue, bInit, (flags AND VisuElems.Visu_InputFlags.Password) = 1, 'O'); END_IF, VisuElemId=-1
    hotkey HotkeyInput Id=481111834624, Key=KeyDown=True, KeyName=P, ActionToExecute=Action=STSnippet=IF bShift THEN VisuDlg_CheckedAppend(stOutputValue, stVariableValue, bInit, (flags AND VisuElems.Visu_InputFlags.Password) = 1, 'p'); ELSE VisuDlg_CheckedAppend(stOutputValue, stVariableValue, bInit, (flags AND VisuElems.Visu_InputFlags.Password) = 1, 'P'); END_IF, VisuElemId=-1
    hotkey HotkeyInput Id=481112883200, Key=KeyDown=True, KeyName=A, ActionToExecute=Action=STSnippet=IF bShift THEN VisuDlg_CheckedAppend(stOutputValue, stVariableValue, bInit, (flags AND VisuElems.Visu_InputFlags.Password) = 1, 'a'); ELSE VisuDlg_CheckedAppend(stOutputValue, stVariableValue, bInit, (flags AND VisuElems.Visu_InputFlags.Password) = 1, 'A'); END_IF, VisuElemId=-1
    hotkey HotkeyInput Id=481113931776, Key=KeyDown=True, KeyName=S, ActionToExecute=Action=STSnippet=IF bShift THEN VisuDlg_CheckedAppend(stOutputValue, stVariableValue, bInit, (flags AND VisuElems.Visu_InputFlags.Password) = 1, 's'); ELSE VisuDlg_CheckedAppend(stOutputValue, stVariableValue, bInit, (flags AND VisuElems.Visu_InputFlags.Password) = 1, 'S'); END_IF, VisuElemId=-1
    hotkey HotkeyInput Id=481114980352, Key=KeyDown=True, KeyName=D, ActionToExecute=Action=STSnippet=IF bShift THEN VisuDlg_CheckedAppend(stOutputValue, stVariableValue, bInit, (flags AND VisuElems.Visu_InputFlags.Password) = 1, 'd'); ELSE VisuDlg_CheckedAppend(stOutputValue, stVariableValue, bInit, (flags AND VisuElems.Visu_InputFlags.Password) = 1, 'D'); END_IF, VisuElemId=-1
    hotkey HotkeyInput Id=481116028928, Key=KeyDown=True, KeyName=F, ActionToExecute=Action=STSnippet=IF bShift THEN VisuDlg_CheckedAppend(stOutputValue, stVariableValue, bInit, (flags AND VisuElems.Visu_InputFlags.Password) = 1, 'f'); ELSE VisuDlg_CheckedAppend(stOutputValue, stVariableValue, bInit, (flags AND VisuElems.Visu_InputFlags.Password) = 1, 'F'); END_IF, VisuElemId=-1
    hotkey HotkeyInput Id=481117077504, Key=KeyDown=True, KeyName=G, ActionToExecute=Action=STSnippet=IF bShift THEN VisuDlg_CheckedAppend(stOutputValue, stVariableValue, bInit, (flags AND VisuElems.Visu_InputFlags.Password) = 1, 'g'); ELSE VisuDlg_CheckedAppend(stOutputValue, stVariableValue, bInit, (flags AND VisuElems.Visu_InputFlags.Password) = 1, 'G'); END_IF, VisuElemId=-1
    hotkey HotkeyInput Id=481118126080, Key=KeyDown=True, KeyName=H, ActionToExecute=Action=STSnippet=IF bShift THEN VisuDlg_CheckedAppend(stOutputValue, stVariableValue, bInit, (flags AND VisuElems.Visu_InputFlags.Password) = 1, 'h'); ELSE VisuDlg_CheckedAppend(stOutputValue, stVariableValue, bInit, (flags AND VisuElems.Visu_InputFlags.Password) = 1, 'H'); END_IF, VisuElemId=-1
    hotkey HotkeyInput Id=481119174656, Key=KeyDown=True, KeyName=J, ActionToExecute=Action=STSnippet=IF bShift THEN VisuDlg_CheckedAppend(stOutputValue, stVariableValue, bInit, (flags AND VisuElems.Visu_InputFlags.Password) = 1, 'j'); ELSE VisuDlg_CheckedAppend(stOutputValue, stVariableValue, bInit, (flags AND VisuElems.Visu_InputFlags.Password) = 1, 'J'); END_IF, VisuElemId=-1
    hotkey HotkeyInput Id=481120223232, Key=KeyDown=True, KeyName=K, ActionToExecute=Action=STSnippet=IF bShift THEN VisuDlg_CheckedAppend(stOutputValue, stVariableValue, bInit, (flags AND VisuElems.Visu_InputFlags.Password) = 1, 'k'); ELSE VisuDlg_CheckedAppend(stOutputValue, stVariableValue, bInit, (flags AND VisuElems.Visu_InputFlags.Password) = 1, 'K'); END_IF, VisuElemId=-1
    hotkey HotkeyInput Id=481121271808, Key=KeyDown=True, KeyName=L, ActionToExecute=Action=STSnippet=IF bShift THEN VisuDlg_CheckedAppend(stOutputValue, stVariableValue, bInit, (flags AND VisuElems.Visu_InputFlags.Password) = 1, 'l'); ELSE VisuDlg_CheckedAppend(stOutputValue, stVariableValue, bInit, (flags AND VisuElems.Visu_InputFlags.Password) = 1, 'L'); END_IF, VisuElemId=-1
    hotkey HotkeyInput Id=481122320384, Key=KeyDown=True, KeyName=Z, ActionToExecute=Action=STSnippet=IF bShift THEN VisuDlg_CheckedAppend(stOutputValue, stVariableValue, bInit, (flags AND VisuElems.Visu_InputFlags.Password) = 1, 'z'); ELSE VisuDlg_CheckedAppend(stOutputValue, stVariableValue, bInit, (flags AND VisuElems.Visu_InputFlags.Password) = 1, 'Z'); END_IF, VisuElemId=-1
    hotkey HotkeyInput Id=481123368960, Key=KeyDown=True, KeyName=X, ActionToExecute=Action=STSnippet=IF bShift THEN VisuDlg_CheckedAppend(stOutputValue, stVariableValue, bInit, (flags AND VisuElems.Visu_InputFlags.Password) = 1, 'x'); ELSE VisuDlg_CheckedAppend(stOutputValue, stVariableValue, bInit, (flags AND VisuElems.Visu_InputFlags.Password) = 1, 'X'); END_IF, VisuElemId=-1
    hotkey HotkeyInput Id=481124417536, Key=KeyDown=True, KeyName=C, ActionToExecute=Action=STSnippet=IF bShift THEN VisuDlg_CheckedAppend(stOutputValue, stVariableValue, bInit, (flags AND VisuElems.Visu_InputFlags.Password) = 1, 'c'); ELSE VisuDlg_CheckedAppend(stOutputValue, stVariableValue, bInit, (flags AND VisuElems.Visu_InputFlags.Password) = 1, 'C'); END_IF, VisuElemId=-1
    hotkey HotkeyInput Id=481125466112, Key=KeyDown=True, KeyName=V, ActionToExecute=Action=STSnippet=IF bShift THEN VisuDlg_CheckedAppend(stOutputValue, stVariableValue, bInit, (flags AND VisuElems.Visu_InputFlags.Password) = 1, 'v'); ELSE VisuDlg_CheckedAppend(stOutputValue, stVariableValue, bInit, (flags AND VisuElems.Visu_InputFlags.Password) = 1, 'V'); END_IF, VisuElemId=-1
    hotkey HotkeyInput Id=481126514688, Key=KeyDown=True, KeyName=B, ActionToExecute=Action=STSnippet=IF bShift THEN VisuDlg_CheckedAppend(stOutputValue, stVariableValue, bInit, (flags AND VisuElems.Visu_InputFlags.Password) = 1, 'b'); ELSE VisuDlg_CheckedAppend(stOutputValue, stVariableValue, bInit, (flags AND VisuElems.Visu_InputFlags.Password) = 1, 'B'); END_IF, VisuElemId=-1
    hotkey HotkeyInput Id=481127563264, Key=KeyDown=True, KeyName=N, ActionToExecute=Action=STSnippet=IF bShift THEN VisuDlg_CheckedAppend(stOutputValue, stVariableValue, bInit, (flags AND VisuElems.Visu_InputFlags.Password) = 1, 'n'); ELSE VisuDlg_CheckedAppend(stOutputValue, stVariableValue, bInit, (flags AND VisuElems.Visu_InputFlags.Password) = 1, 'N'); END_IF, VisuElemId=-1
    hotkey HotkeyInput Id=481128611840, Key=KeyDown=True, KeyName=M, ActionToExecute=Action=STSnippet=IF bShift THEN VisuDlg_CheckedAppend(stOutputValue, stVariableValue, bInit, (flags AND VisuElems.Visu_InputFlags.Password) = 1, 'm'); ELSE VisuDlg_CheckedAppend(stOutputValue, stVariableValue, bInit, (flags AND VisuElems.Visu_InputFlags.Password) = 1, 'M'); END_IF, VisuElemId=-1
    hotkey HotkeyInput Id=481129660416, Key=KeyDown=True, KeyName=COMMA, ActionToExecute=Action=STSnippet=IF bShift THEN VisuDlg_CheckedAppend(stOutputValue, stVariableValue, bInit, (flags AND VisuElems.Visu_InputFlags.Password) = 1, ','); ELSE VisuDlg_CheckedAppend(stOutputValue, stVariableValue, bInit, (flags AND VisuElems.Visu_InputFlags.Password) = 1, '.'); END_IF, VisuElemId=-1
    hotkey HotkeyInput Id=481131757568, Key=KeyDown=True, KeyName=NUM1, ActionToExecute=Action=STSnippet=VisuDlg_CheckedAppend(stOutputValue, stVariableValue, bInit, (flags AND VisuElems.Visu_InputFlags.Password) = 1, '1');, VisuElemId=-1
    hotkey HotkeyInput Id=481132806144, Key=KeyDown=True, KeyName=NUM2, ActionToExecute=Action=STSnippet=VisuDlg_CheckedAppend(stOutputValue, stVariableValue, bInit, (flags AND VisuElems.Visu_InputFlags.Password) = 1, '2');, VisuElemId=-1
    hotkey HotkeyInput Id=481133854720, Key=KeyDown=True, KeyName=NUM3, ActionToExecute=Action=STSnippet=VisuDlg_CheckedAppend(stOutputValue, stVariableValue, bInit, (flags AND VisuElems.Visu_InputFlags.Password) = 1, '3');, VisuElemId=-1
    hotkey HotkeyInput Id=481134903296, Key=KeyDown=True, KeyName=NUM4, ActionToExecute=Action=STSnippet=VisuDlg_CheckedAppend(stOutputValue, stVariableValue, bInit, (flags AND VisuElems.Visu_InputFlags.Password) = 1, '4');, VisuElemId=-1
    hotkey HotkeyInput Id=481135951872, Key=KeyDown=True, KeyName=NUM5, ActionToExecute=Action=STSnippet=VisuDlg_CheckedAppend(stOutputValue, stVariableValue, bInit, (flags AND VisuElems.Visu_InputFlags.Password) = 1, '5');, VisuElemId=-1
    hotkey HotkeyInput Id=481137000448, Key=KeyDown=True, KeyName=NUM6, ActionToExecute=Action=STSnippet=VisuDlg_CheckedAppend(stOutputValue, stVariableValue, bInit, (flags AND VisuElems.Visu_InputFlags.Password) = 1, '6');, VisuElemId=-1
    hotkey HotkeyInput Id=481138049024, Key=KeyDown=True, KeyName=NUM7, ActionToExecute=Action=STSnippet=VisuDlg_CheckedAppend(stOutputValue, stVariableValue, bInit, (flags AND VisuElems.Visu_InputFlags.Password) = 1, '7');, VisuElemId=-1
    hotkey HotkeyInput Id=481139097600, Key=KeyDown=True, KeyName=NUM8, ActionToExecute=Action=STSnippet=VisuDlg_CheckedAppend(stOutputValue, stVariableValue, bInit, (flags AND VisuElems.Visu_InputFlags.Password) = 1, '8');, VisuElemId=-1
    hotkey HotkeyInput Id=481140146176, Key=KeyDown=True, KeyName=NUM9, ActionToExecute=Action=STSnippet=VisuDlg_CheckedAppend(stOutputValue, stVariableValue, bInit, (flags AND VisuElems.Visu_InputFlags.Password) = 1, '9');, VisuElemId=-1
    hotkey HotkeyInput Id=481141194752, Key=KeyDown=True, KeyName=NUM0, ActionToExecute=Action=STSnippet=VisuDlg_CheckedAppend(stOutputValue, stVariableValue, bInit, (flags AND VisuElems.Visu_InputFlags.Password) = 1, '0');, VisuElemId=-1
END_VISUALIZATION

// ---- VISUs/Kierwonica.TcVIS
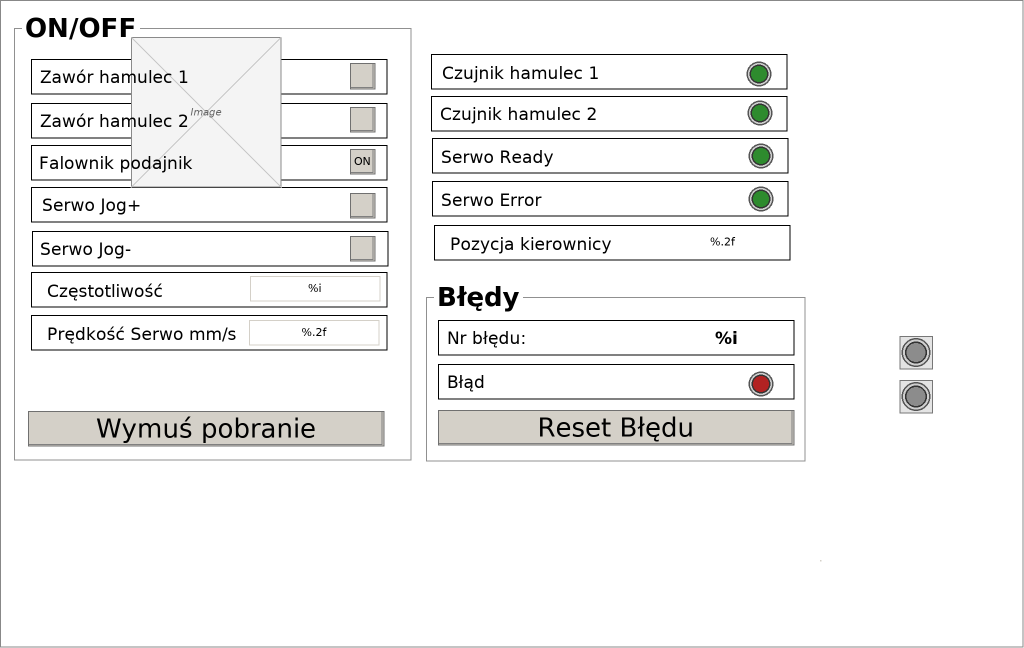
VISUALIZATION Kierwonica  // 1024x648
    Rectangle (31,59 356x35)
    Rectangle (31,103 356x35)
    Rectangle (31,145 356x35)
    Rectangle (31,272 356x35)
    Rectangle (32,231 356x35)
    Rectangle (31,187 356x35)
    GroupBox (14,20 397x440), "ON/OFF"
        Rectangle (17,295 356x35)
        Button (336,173 25x25)
            tap GVL_HMI.bHmiJogF
        Button (336,216 25x25)
            tap GVL_HMI.bHmiJogB
        Textfield (236,256 130x25), "%i", text variable: GVL_HMI.iFreqKierownicaMan
            OnMouseClick: write the text variable via Edit
        Button (336,129 25x25), "ON", colour toggle: GVL_GLOBAL.falownik_podajnik_kier_cewka
            tap GVL_HMI.przycisk_falownik_podajnik_kier
        Button (336,87 25x25), colour toggle: GVL_GLOBAL.zaw_ham2_kier_cewka
            tap GVL_HMI.przycisk_zaw_ham2_kier
        Button (336,43 25x26), colour toggle: GVL_GLOBAL.zaw_ham1_kier_cewka
            tap GVL_HMI.przycisk_zaw_ham1_kier
        Image (117,17 150x150)
        Button (14,391 356x35), "Wymuś pobranie"
            OnMouseDown: execute { GVL_HMI.Wymus_pobranie:=TRUE; }
    Rectangle (431,54 356x35)
    Label (437,57 230x30)
    Rectangle (431,96 356x35)
    Label (437,99 239x30), "Czujnik hamulec 2"
    Lamp1 (746,99 28x28), variable: GVL_IO_K.b4B6, style: Lamp-Lamp1-Green
    Lamp1 (745,60 28x28), variable: GVL_IO_K.b4B7, style: Lamp-Lamp1-Green
    Label (439,58 239x30), "Czujnik hamulec 1"
    Rectangle (432,138 356x35)
    Rectangle (432,181 356x35)
    Label (37,101 239x30)
    Label (37,106 209x30), "Zawór hamulec 2"
    Label (37,62 209x30), "Zawór hamulec 1"
    Label (36,148 209x30), "Falownik podajnik"
    Label (44,276 209x30), "Częstotliwość"
    Label (438,142 239x30), "Serwo Ready"
    Lamp1 (747,142 28x28), variable: PRG_Kierownica.S_K_Power.Status, style: Lamp-Lamp1-Green
    Label (438,185 239x30), "Serwo Error"
    Lamp1 (747,185 28x28), variable: PRG_Kierownica.S_K_Power.Error, style: Lamp-Lamp1-Green
    Rectangle (434,225 356x35)
    Label (447,229 209x30), "Pozycja kierownicy"
    Textfield (662,227 121x30), "%.2f", text variable: GVL_AXIS.stAxis2.NcToPlc.ActPos
    Label (39,190 209x30), "Serwo Jog+"
    Label (37,234 209x30), "Serwo Jog-"
    PushSwitch (897,380 38x33), behaviour: TOGGLE, style: Switch-PushSwitch-Gray
    PushSwitch (897,336 38x33), behaviour: TOGGLE, style: Switch-PushSwitch-Gray
    Textfield (249,320 130x25), "%.2f", text variable: gvl_hmi.J_Vel
        OnMouseClick: write the text variable via Edit
    Label (44,319 209x30), "Prędkość Serwo mm/s"
    Textfield (820,560 1x1)
    GroupBox (426,289 379x172), "Błędy"
        Rectangle (12,31 356x35)
        Label (18,34 209x30), "Nr błędu:"
        Rectangle (12,75 356x35)
        Label (18,78 209x30), "Błąd"
        Button (12,121 356x35), "Reset Błędu"
            tap GVL_HMI.ErrorResetKier
        Lamp1 (321,81 28x28), variable: GVL_GLOBAL.Error_pakowania, style: Lamp-Lamp1-Red
        Textfield (240,34 121x30), "%i", text variable: GVL_GLOBAL.Error_numb_kier
END_VISUALIZATION

// ---- VISUs/mssgbox.TcVIS
VISUALIZATION mssgbox  // 200x100
END_VISUALIZATION

// ---- VISUs/PH_AxisOnline.TcVIS
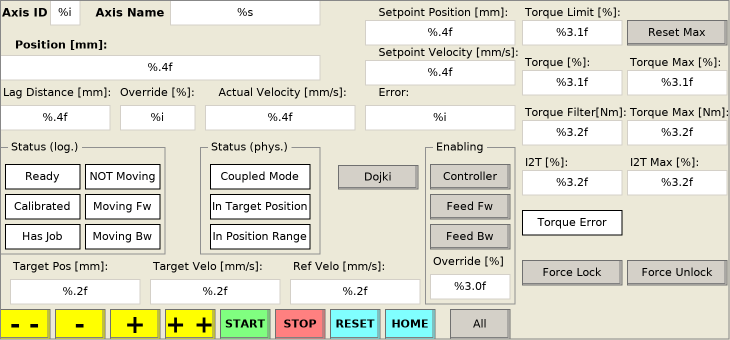
VISUALIZATION PH_AxisOnline  // 730x340
//==================================================================================================
//							Beckhoff Automation Poland
//									18.04.2018
//	Wizualizacja dla Axis Online
//  v1.0	|| TC v 3.1.4022.16		|| - pierwsza wersja
//==================================================================================================
VAR_IN_OUT
	stMcAxisOnline			: ST_McAxisOnline;	
END_VAR
    Frame (0,0 520x340)
        shows PH_NcAxis(stMcAxisOnline := stMcAxisOnline)
    Frame (520,0 210x340)
        shows PH_Motor(stMcAxisOnline := stMcAxisOnline)
END_VISUALIZATION

// ---- VISUs/PH_AxisOnline_1.TcVIS
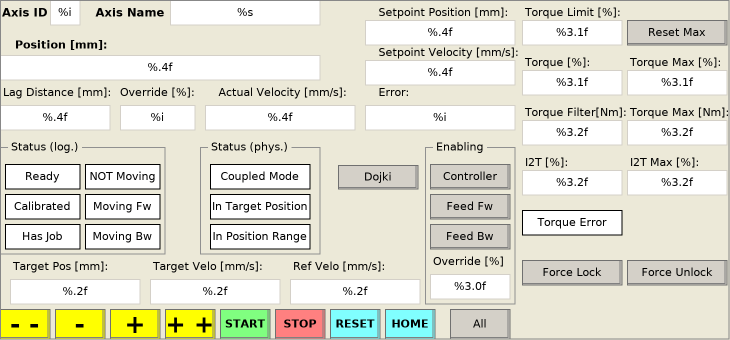
VISUALIZATION PH_AxisOnline_1  // 730x340
//==================================================================================================
//							Beckhoff Automation Poland
//									18.04.2018
//	Wizualizacja dla Axis Online
//  v1.0	|| TC v 3.1.4022.16		|| - pierwsza wersja
//==================================================================================================
VAR_IN_OUT
	stMcAxisOnline			: ST_McAxisOnline;	
END_VAR
    Frame (0,0 520x340)
        shows PH_NcAxis(stMcAxisOnline := stMcAxisOnline)
    Frame (520,0 210x340)
        shows PH_Motor(stMcAxisOnline := stMcAxisOnline)
END_VISUALIZATION

// ---- VISUs/PH_Motor.TcVIS
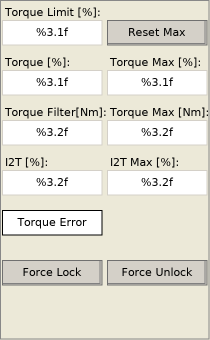
VISUALIZATION PH_Motor  // 210x340
//==================================================================================================
//							Beckhoff Automation Poland
//									18.04.2018
//	Wizualizacja dla Axis Online
//  v1.0	|| TC v 3.1.4022.16		|| - pierwsza wersja
//==================================================================================================
VAR_IN_OUT
	stMcAxisOnline			: ST_McAxisOnline;	
END_VAR
    Button (107,20 100x25), "Reset Max"
        tap stMcAxisOnline.stMotorMonitoring.bReset
    Group (2,0 100x45)
        Textfield (0,20 100x25), "%3.1f", text variable: stMcAxisOnline.stMotorMonitoring.rTorqueLimit
            OnMouseClick: write the text variable via InputWithLimits, min 0, max 500
        Label (0,0 100x25), "Torque Limit [%]:"
    Rectangle (2,210 100x25), "Torque Error", colour toggle: stMcAxisOnline.stMotorMonitoring.bError
    Group (2,100 100x45)
        Textfield (0,20 100x25), "%3.2f", text variable: stMcAxisOnline.stMotorMonitoring.rTorqueF, colour toggle: stMcAxisOnline.stMotorMonitoring.bWarning
        Label (0,0 100x25), "Torque Filter[Nm]:"
    Group (107,100 100x45)
        Textfield (0,20 100x25), "%3.2f", text variable: stMcAxisOnline.stMotorMonitoring.rTorqueMax
        Label (0,0 100x25), "Torque Max [Nm]:"
    Group (2,150 100x45)
        Label (0,0 100x25), "I2T [%]:"
        Textfield (0,20 100x25), "%3.2f", text variable: stMcAxisOnline.stMotorMonitoring.rI2T
    Group (107,150 100x45)
        Label (0,0 100x25), "I2T Max [%]:"
        Textfield (0,20 100x25), "%3.2f", text variable: stMcAxisOnline.stMotorMonitoring.rI2TMax
    Button (2,260 100x25), "Force Lock"
        tap stMcAxisOnline.stHoldingBrake.bForceLock
    Button (107,260 100x25), "Force Unlock"
        tap stMcAxisOnline.stHoldingBrake.bForceUnlock
    Group (2,50 100x45)
        Textfield (0,20 100x25), "%3.1f", text variable: stMcAxisOnline.stMotorMonitoring.rTorquePerc, colour toggle: stMcAxisOnline.stMotorMonitoring.bWarning
        Label (0,0 100x25), "Torque [%]:"
    Group (107,50 100x45)
        Textfield (0,20 100x25), "%3.1f", text variable: stMcAxisOnline.stMotorMonitoring.rTorquePercMax
        Label (0,0 100x25), "Torque Max [%]:"
END_VISUALIZATION

// ---- VISUs/PH_NcAxis.TcVIS
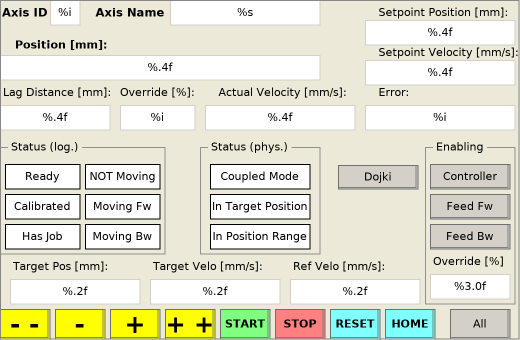
VISUALIZATION PH_NcAxis  // 520x340
VAR_IN_OUT
	stMcAxisOnline			: ST_McAxisOnline;	
END_VAR
    Group (0,0 320x25)
        Label (0,0 50x25), "Axis ID"
        Textfield (50,0 30x25), "%i", text variable: stMcAxisOnline.stStatus.dwAxisId
        Label (90,0 80x25), "Axis Name"
        Textfield (170,0 150x25), "%s", text variable: stMcAxisOnline.stStatus.sAxisName
    GroupBox (425,139 90x165), "Enabling"
        Button (5,25 80x25), "Controller", pressed state: stMcAxisOnline.mcPower.bEnable
            toggle stMcAxisOnline.mcPower.bEnable
        Button (5,85 80x25), "Feed Bw", pressed state: stMcAxisOnline.mcPower.bEnable_Negative
            toggle stMcAxisOnline.mcPower.bEnable_Negative
        Button (5,55 80x25), "Feed Fw", pressed state: stMcAxisOnline.mcPower.bEnable_Positive
            toggle stMcAxisOnline.mcPower.bEnable_Positive
        Textfield (5,135 80x25), "%3.0f", text variable: stMcAxisOnline.mcPower.lrOverride
            OnMouseClick: write the text variable via InputWithLimits, min 0, max 100
        Label (5,110 80x25), "Override [%]"
    Group (0,30 320x50)
        Textfield (0,25 320x25), "%.4f", text variable: stMcAxisOnline.stStatus.lrActPos
        Label (0,0 139x30), "Position [mm]:"
    GroupBox (200,139 120x115), "Status (phys.)"
        Rectangle (10,25 100x25), "Coupled Mode", colour toggle: stMcAxisOnline.stStatus.stAxisStatus.ProtectedMode
        Rectangle (10,55 100x25), "In Target Position", colour toggle: stMcAxisOnline.stStatus.stAxisStatus.InTargetPosition
        Rectangle (10,85 100x25), "In Position Range", colour toggle: stMcAxisOnline.stStatus.stAxisStatus.InPositionArea
    GroupBox (0,139 165x115), "Status (log.)"
        Rectangle (5,55 75x25), "Calibrated", colour toggle: stMcAxisOnline.stStatus.stAxisStatus.Homed
        Rectangle (5,85 75x25), "Has Job", colour toggle: stMcAxisOnline.stStatus.stAxisStatus.HasJob
        Rectangle (85,25 75x25), "NOT Moving", colour toggle: stMcAxisOnline.stStatus.stAxisStatus.NotMoving
        Rectangle (85,55 75x25), "Moving Fw", colour toggle: stMcAxisOnline.stStatus.stAxisStatus.PositiveDirection
        Rectangle (85,85 75x25), "Moving Bw", colour toggle: stMcAxisOnline.stStatus.stAxisStatus.NegativeDirection
        Rectangle (5,25 75x25), "Ready", colour toggle: stMcAxisOnline.stStatus.stAxisStatus.Operational
    Group (365,0 150x130)
        Label (0,0 150x25), "Setpoint Position [mm]:"
        Textfield (0,20 150x25), "%.4f", text variable: stMcAxisOnline.stStatus.lrSetPos
        Label (0,40 150x25), "Setpoint Velocity [mm/s]:"
        Textfield (0,60 150x25), "%.4f", text variable: stMcAxisOnline.stStatus.lrSetVelo
        Label (0,80 150x25), "Error:"
        Textfield (0,105 150x25), "%i", text variable: stMcAxisOnline.stStatus.udiNcErrorCode, colour toggle: stMcAxisOnline.stStatus.udiNcErrorCode>0
    Group (205,80 150x50)
        Label (0,0 150x25), "Actual Velocity [mm/s]:"
        Textfield (0,25 150x25), "%.4f", text variable: stMcAxisOnline.stStatus.lrActVelo
    Group (0,80 110x50)
        Label (0,0 110x25), "Lag Distance [mm]:"
        Textfield (0,25 110x25), "%.4f", text variable: stMcAxisOnline.stStatus.lrPosDiff
    Group (120,80 75x50)
        Label (0,0 75x25), "Override [%]:"
        Textfield (0,25 75x25), "%i", text variable: stMcAxisOnline.mcPower.lrOverride
    Label (290,254 130x25), "Ref Velo [mm/s]:"
    Textfield (290,279 130x25), "%.2f", text variable: stMcAxisOnline.stAxisParameter.fDriveVeloReferenz
        OnMouseClick: write the text variable via Edit
    Label (10,254 130x25), "Target Pos [mm]:"
    Textfield (10,279 130x25), "%.2f", text variable: stMcAxisOnline.mcMoveAbsolute.lrPosition
        OnMouseClick: write the text variable via Edit
    Label (150,254 130x25), "Target Velo [mm/s]:"
    Textfield (150,279 130x25), "%.2f", text variable: stMcAxisOnline.mcMoveAbsolute.lrVelocity
        OnMouseClick: write the text variable via Edit
    Button (450,309 60x30), "All"
        OnMouseClick: execute {
            stMcAxisOnline.mcPower.bEnable				:= TRUE;
            stMcAxisOnline.mcPower.bEnable_Positive		:= TRUE;
            stMcAxisOnline.mcPower.bEnable_Negative		:= TRUE;
            stMcAxisOnline.mcPower.lrOverride			:= 100.0;
        }
    Group (0,309 435x30)
        Button (220,0 50x30), "START"
            tap stMcAxisOnline.mcMoveAbsolute.bExecute
        Button (275,0 50x30), "STOP"
            tap stMcAxisOnline.mcStop.bExecute
        Button (385,0 50x30), "HOME"
            tap stMcAxisOnline.mcHome.bExecute
        Button (330,0 50x30), "RESET"
            tap stMcAxisOnline.mcReset.bExecute
        Button (110,0 50x30), "+"
            tap stMcAxisOnline.mcJog.bSlowForward
        Button (165,0 50x30), "+ +"
            tap stMcAxisOnline.mcJog.bFastForward
        Button (55,0 50x30), "-"
            tap stMcAxisOnline.mcJog.bSlowBackward
        Button (0,0 50x30), "- -"
            tap stMcAxisOnline.mcJog.bFastBackward
    Button (338,165 80x24), "Dojki", pressed state: GVL_HMI.bDojkiM
        toggle GVL_HMI.bDojkiM
END_VISUALIZATION

// ---- VISUs/Ploter.TcVIS
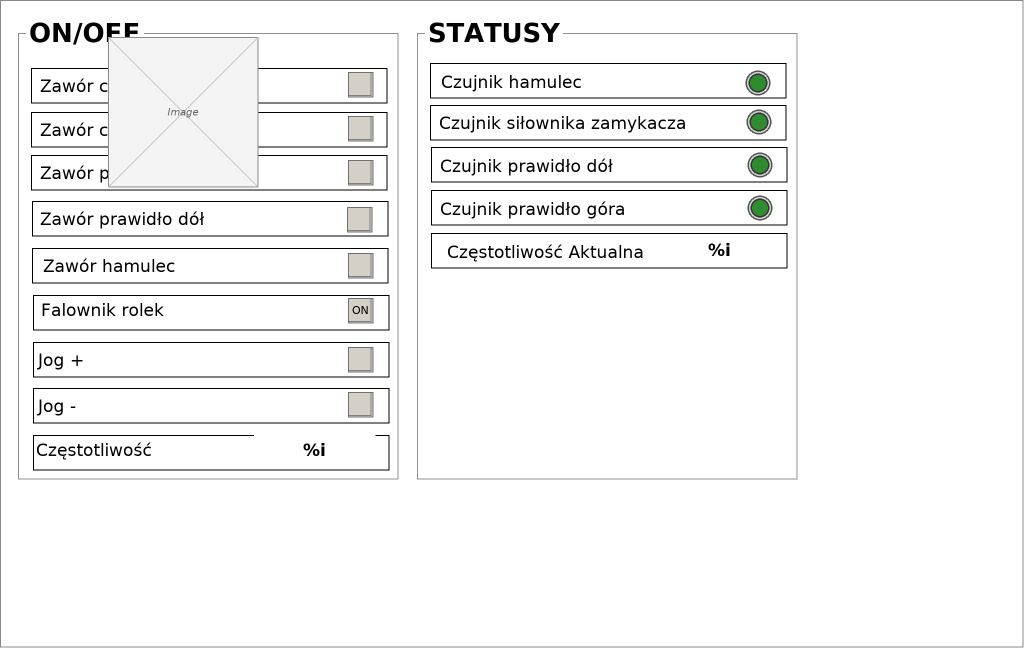
VISUALIZATION Ploter  // 1024x648
    Rectangle (31,155 356x35)
    Label (37,158 208x30), "Zawór prawidło"
    GroupBox (18,25 380x454), "ON/OFF"
        Rectangle (13,43 356x35)
        Rectangle (13,87 356x35)
        Rectangle (15,270 356x35)
        Rectangle (14,223 356x35)
        Label (19,85 239x30)
        Label (19,90 209x30), "Zawór chwytaka 2"
        Label (19,46 209x30), "Zawór chwytaka 1"
        Label (22,226 209x30), "Zawór hamulec"
        Label (20,270 209x30), "Falownik rolek"
        Rectangle (15,410 356x35)
        Label (15,410 216x30), "Częstotliwość"
        Textfield (236,410 121x30), "%i", text variable: GVL_HMI.iWydajnosc
        Button (330,228 25x25), colour toggle: GVL_GLOBAL.zaw_hamulec_cewka
            tap GVL_HMI.przycisk_zaw_hamulec
        Button (330,273 25x25), "ON", colour toggle: GVL_GLOBAL.falownik_rolek_cewka
            tap GVL_HMI.przycisk_falownik_rolek
        Button (330,91 25x25), colour toggle: GVL_GLOBAL.zaw_chwyt2_cewka
            tap GVL_HMI.przycisk_zaw_chwyt2
        Button (330,47 25x25), colour toggle: GVL_GLOBAL.zaw_chwyt1_cewka
            tap GVL_HMI.przycisk_zaw_chwyt1
        Rectangle (14,176 356x35)
        Button (330,135 25x25), colour toggle: GVL_GLOBAL.zaw_prawidlo_cewka
            tap GVL_HMI.przycisk_zaw_prawidlo
        Button (329,182 25x25), colour toggle: GVL_GLOBAL.zaw_prawidlo_dol_cewka
            tap GVL_HMI.przycisk_zaw_prawdidlo_dol
        Rectangle (15,317 356x35)
        Rectangle (15,363 356x35)
        Label (17,320 209x30), "Jog +"
        Label (17,366 209x30), "Jog -"
        Button (330,322 25x25), colour toggle: GVL_GLOBAL.zaw_hamulec_cewka
            tap GVL_HMI.bHmiPlotCCw
        Button (330,367 25x25), colour toggle: GVL_GLOBAL.zaw_hamulec_cewka
            tap GVL_HMI.bHmiPlotCw
    Image (108,37 150x150)
    GroupBox (417,25 380x454), "STATUSY"
        Rectangle (13,38 356x35)
        Label (19,41 230x30)
        Rectangle (13,80 356x35)
        Label (19,83 239x30), "Czujnik siłownika zamykacza"
        Lamp1 (328,83 28x28), variable: GVL_IO_P.b3B1, style: Lamp-Lamp1-Green
        Lamp1 (327,44 28x28), variable: GVL_IO_P.b5B1, style: Lamp-Lamp1-Green
        Label (21,42 239x30), "Czujnik hamulec"
        Rectangle (14,122 356x35)
        Rectangle (14,165 356x35)
        Rectangle (14,208 356x35)
        Label (27,212 209x30), "Częstotliwość Aktualna"
        Textfield (242,210 121x30), "%i", text variable: GVL_HMI.iWydajnosc
    Label (437,151 239x30), "Czujnik prawidło dół"
    Lamp1 (746,151 28x28), variable: GVL_IO_P.b2B1, style: Lamp-Lamp1-Green
    Label (437,194 239x30), "Czujnik prawidło góra"
    Lamp1 (746,194 28x28), variable: GVL_IO_P.b6B1, style: Lamp-Lamp1-Green
    Label (37,204 212x30), "Zawór prawidło dół"
END_VISUALIZATION

// ---- VISUs/Statystyki.TcVIS
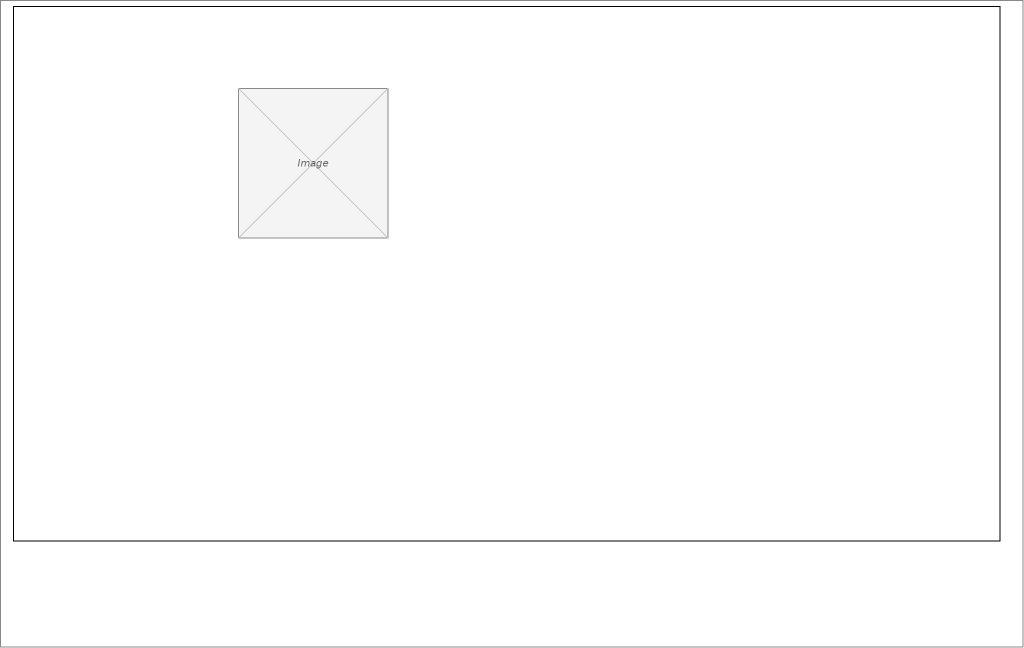
VISUALIZATION Statystyki  // 1024x648
    Rectangle (13,6 987x535)
    Image (238,88 150x150)
END_VISUALIZATION

// ---- VISUs/Serwis.TcVIS
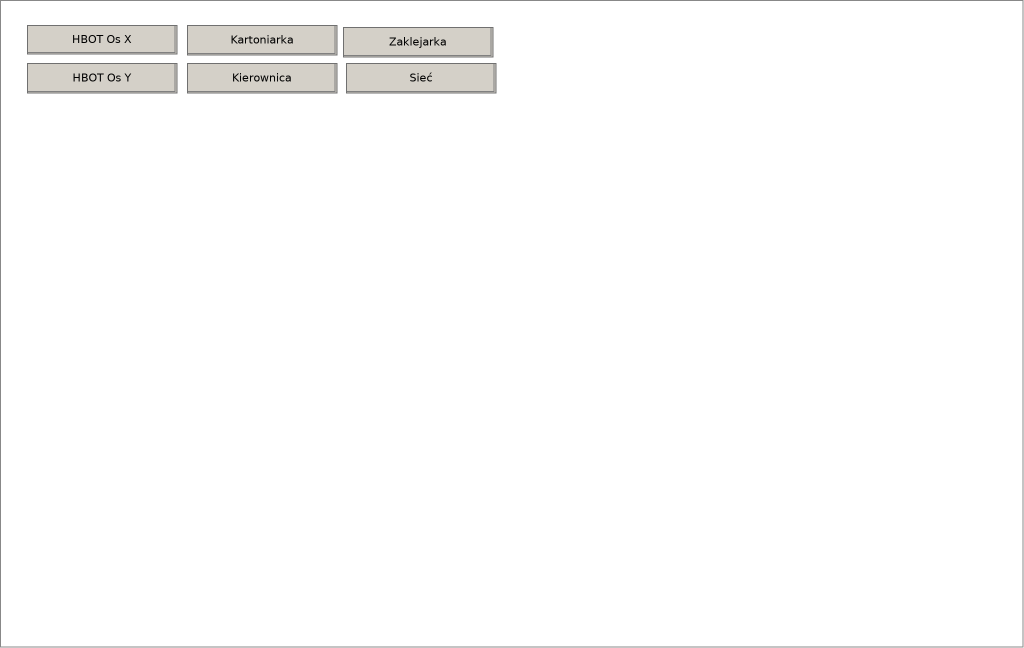
VISUALIZATION Serwis  // 1024x648
    Button (27,25 150x29), "HBOT Os X", colour toggle: GVL_HMI.strona_1=2
        OnMouseDown: FrameSelectionChange Selection=SelectedFrame=9731c5c5-429f-486e-9358-6f2f3bdb5ae0, GlobSel=AssignType=Directly, SelType=Locally
        OnMouseDown: execute { GVL_HMI.strona_1:=2; }
    Button (187,25 150x30), "Kartoniarka"
    Button (343,27 150x30), "Zaklejarka"
    Button (187,63 150x30), "Kierownica"
    Button (346,63 150x30), "Sieć"
    Button (27,63 150x30), "HBOT Os Y", colour toggle: GVL_HMI.strona_1=1
        OnMouseDown: FrameSelectionChange Selection=SelectedFrame=9731c5c5-429f-486e-9358-6f2f3bdb5ae0, Selection=1, GlobSel=AssignType=Directly, SelType=Locally
        OnMouseDown: execute { GVL_HMI.strona_1:=1; }
END_VISUALIZATION

// ---- VISUs/Visualization.TcVIS
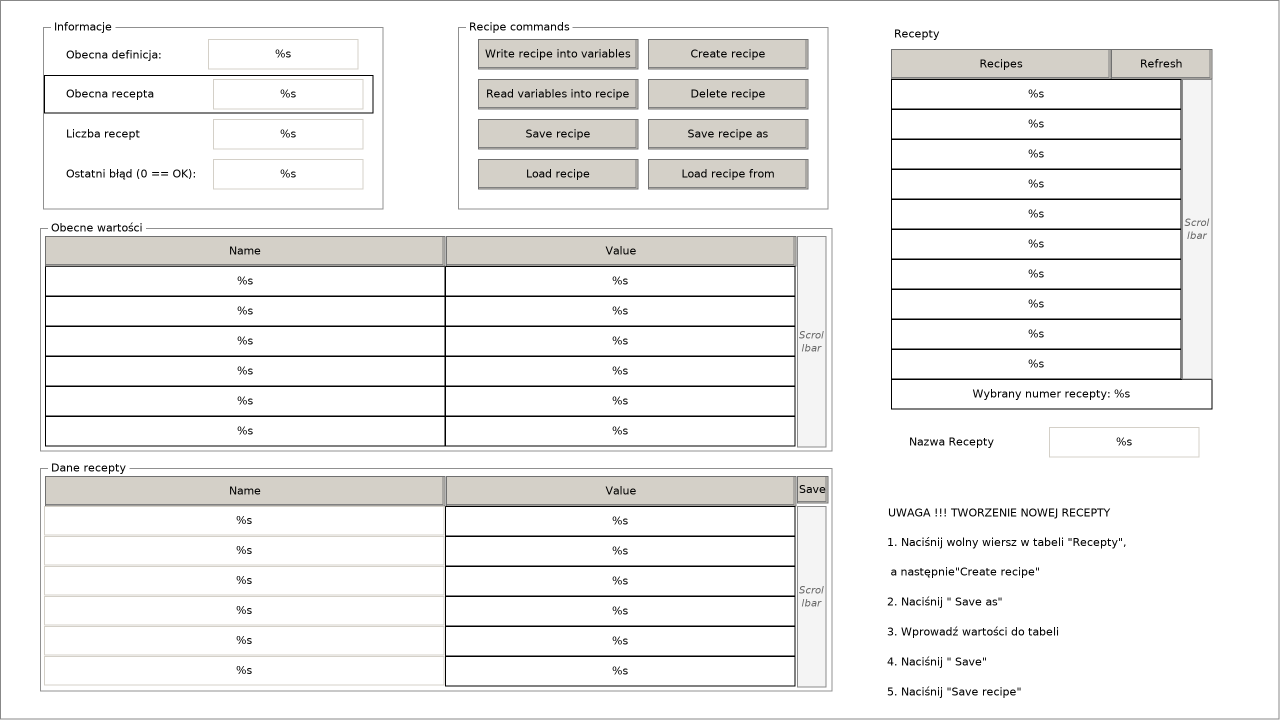
VISUALIZATION Visualization  // 1280x720
    GroupBox (40,220 792x231), "Obecne wartości"
        Rectangle (5,46 400x30), "%s", text variable: GVL_RecipeTable.aVariableNames[GVL_RecipeTable.nVariableIndex], input disabled if: TRUE
        Rectangle (5,76 400x30), "%s", text variable: GVL_RecipeTable.aVariableNames[GVL_RecipeTable.nVariableIndex+1], input disabled if: TRUE
        Rectangle (5,136 400x30), "%s", text variable: GVL_RecipeTable.aVariableNames[GVL_RecipeTable.nVariableIndex+3], input disabled if: TRUE
        Rectangle (5,166 400x30), "%s", text variable: GVL_RecipeTable.aVariableNames[GVL_RecipeTable.nVariableIndex+4], input disabled if: TRUE
        Rectangle (5,196 400x30), "%s", text variable: GVL_RecipeTable.aVariableNames[GVL_RecipeTable.nVariableIndex+5], input disabled if: TRUE
        Rectangle (5,106 400x30), "%s", text variable: GVL_RecipeTable.aVariableNames[GVL_RecipeTable.nVariableIndex+2], input disabled if: TRUE
    GroupBox (40,460 792x231), "Dane recepty"
    GroupBox (43,19 340x190), "Informacje"
        Rectangle (1,56 329x38)
        Textfield (165,20 150x30), "%s", text variable: RecipeManagement.sRecipeDef, input disabled if: TRUE
            OnMouseClick: write the text variable via Default
        Label (20,21 150x30), "Obecna definicja:"
        Label (20,60 150x30), "Obecna recepta"
        Label (20,140 150x30), "Ostatni błąd (0 == OK):"
        Label (20,100 150x30), "Liczba recept"
        Textfield (170,60 150x30), "%s", text variable: RecipeManagement.sRecipe, input disabled if: TRUE
            OnMouseClick: write the text variable via Default
        Textfield (170,140 150x30), "%s", text variable: RecipeManagement.nLastError, input disabled if: TRUE
        Textfield (170,100 150x30), "%s", text variable: RecipeManagement.nRecipeCount, input disabled if: TRUE
    GroupBox (458,19 370x190), "Recipe commands"
        Button (20,20 160x30), "Write recipe into variables"
            OnMouseClick: ExecuteCommand ExecuteCommand=ExecuteCommand=[Command=WriteRecipe, Value=RecipeManagement.sRecipeDef, Value2=RecipeManagement.sRecipe]
        Button (20,60 160x30), "Read variables into recipe"
            OnMouseClick: ExecuteCommand ExecuteCommand=ExecuteCommand=[Command=ReadRecipe, Value=RecipeManagement.sRecipeDef, Value2=RecipeManagement.sRecipe]
            OnMouseClick: execute { RecipeManagement.bReloadValues := TRUE; }
        Button (20,100 160x30), "Save recipe"
            OnMouseClick: ExecuteCommand ExecuteCommand=ExecuteCommand=[Command=SaveRecipe, Value=RecipeManagement.sRecipeDef, Value2=RecipeManagement.sRecipe]
        Button (20,140 160x30), "Load recipe"
            OnMouseClick: ExecuteCommand ExecuteCommand=ExecuteCommand=[Command=LoadRecipe, Value=RecipeManagement.sRecipeDef, Value2=RecipeManagement.sRecipe]
            OnMouseClick: toggle RecipeManagement.bReloadValues
            OnMouseClick: execute {
                GVL_RecipeTable.aCurrentValues[0]:=GVL_Recipe.dl_kartonu;
                GVL_RecipeTable.aCurrentValues[1]:=GVL_Recipe.wys_kartonu;
                GVL_RecipeTable.aCurrentValues[2]:=GVL_Recipe.szer_kartonu;
                GVL_RecipeTable.aCurrentValues[3]:=GVL_Recipe.Poz_X_Odlozenie;
                GVL_RecipeTable.aCurrentValues[4]:=GVL_Recipe.Il_kolumn;
                GVL_RecipeTable.aCurrentValues[5]:=GVL_Recipe.Il_rzedow;
                GVL_RecipeTable.aCurrentValues[6]:=GVL_Recipe.Predk_mag_odlozenie;
                GVL_RecipeTable.aCurrentValues[7]:=GVL_Recipe.Predk_mag_pobranie;
                GVL_RecipeTable.aCurrentValues[8]:=GVL_Recipe.Predk_plot_odlozenie;
                GVL_RecipeTable.aCurrentValues[9]:=GVL_Recipe.Predk_plot_pobranie;
                GVL_RecipeTable.aCurrentValues[10]:=GVL_Recipe.Predk_plot_ruch;
                GVL_RecipeTable.aCurrentValues[11]:=GVL_Recipe.Poz_Z_Odlozenie;
                GVL_RecipeTable.aCurrentValues[12]:=GVL_Recipe.Poz_Z_Pobranie;
            }
            OnMouseClick: execute { GVL_RecipeTable.aCurrentVariableNames:=GVL_RecipeTable.aVariableNames; }
        Button (190,20 160x30), "Create recipe"
            OnMouseClick: ExecuteCommand ExecuteCommand=ExecuteCommand=[Command=CreateRecipe, Value=RecipeManagement.sRecipeDef, Value2=MAIN.sRecipe]
            OnMouseClick: execute { RecipeManagement.bReload := TRUE; }
        Button (190,100 160x30), "Save recipe as"
            OnMouseClick: ExecuteCommand ExecuteCommand=ExecuteCommand=[Command=SaveRecipeAs, Value=RecipeManagement.sRecipeDef, Value2=RecipeManagement.sRecipe]
        Button (190,140 160x30), "Load recipe from"
            OnMouseClick: ExecuteCommand ExecuteCommand=ExecuteCommand=[Command=LoadRecipeFrom, Value=RecipeManagement.sRecipeDef, Value2=RecipeManagement.sRecipe]
        Button (190,60 160x30), "Delete recipe"
            OnMouseClick: ExecuteCommand ExecuteCommand=ExecuteCommand=[Command=DeleteRecipe, Value=RecipeManagement.sRecipeDef, Value2=RecipeManagement.sRecipe]
            OnMouseClick: execute { RecipeManagement.bInit := TRUE; }
    Button (891,49 220x30), "Recipes"
        OnMouseDown: toggle RecipeManagement.bReload
    Label (891,19 322x30), "Recepty"
    Button (1111,49 101x30), "Refresh"
        OnMouseDown: toggle RecipeManagement.bReload
    Rectangle (891,79 290x30), "%s", text variable: GVL_RecipeTable.aRecipeNames[GVL_RecipeTable.nRecipeIndex], colour toggle: (GVL_RecipeTable.nRecipeSelectionIndex-GVL_RecipeTable.nRecipeIndex) = 0
        OnMouseDown: execute { GVL_RecipeTable.nRecipeSelectionIndex := GVL_RecipeTable.nRecipeIndex; }
    Rectangle (891,109 290x30), "%s", text variable: GVL_RecipeTable.aRecipeNames[GVL_RecipeTable.nRecipeIndex+1], colour toggle: (GVL_RecipeTable.nRecipeSelectionIndex-GVL_RecipeTable.nRecipeIndex) = 1
        OnMouseDown: execute { GVL_RecipeTable.nRecipeSelectionIndex := GVL_RecipeTable.nRecipeIndex + 1; }
    Rectangle (891,139 290x30), "%s", text variable: GVL_RecipeTable.aRecipeNames[GVL_RecipeTable.nRecipeIndex+2], colour toggle: (GVL_RecipeTable.nRecipeSelectionIndex-GVL_RecipeTable.nRecipeIndex) = 2
        OnMouseDown: execute { GVL_RecipeTable.nRecipeSelectionIndex := GVL_RecipeTable.nRecipeIndex + 2; }
    Rectangle (891,169 290x30), "%s", text variable: GVL_RecipeTable.aRecipeNames[GVL_RecipeTable.nRecipeIndex+3], colour toggle: (GVL_RecipeTable.nRecipeSelectionIndex-GVL_RecipeTable.nRecipeIndex) = 3
        OnMouseDown: execute { GVL_RecipeTable.nRecipeSelectionIndex := GVL_RecipeTable.nRecipeIndex + 3; }
    Rectangle (891,199 290x30), "%s", text variable: GVL_RecipeTable.aRecipeNames[GVL_RecipeTable.nRecipeIndex+4], colour toggle: (GVL_RecipeTable.nRecipeSelectionIndex-GVL_RecipeTable.nRecipeIndex) = 4
        OnMouseDown: execute { GVL_RecipeTable.nRecipeSelectionIndex := GVL_RecipeTable.nRecipeIndex + 4; }
    Rectangle (891,229 290x30), "%s", text variable: GVL_RecipeTable.aRecipeNames[GVL_RecipeTable.nRecipeIndex+5], colour toggle: (GVL_RecipeTable.nRecipeSelectionIndex-GVL_RecipeTable.nRecipeIndex) = 5
        OnMouseDown: execute { GVL_RecipeTable.nRecipeSelectionIndex := GVL_RecipeTable.nRecipeIndex + 5; }
    Rectangle (891,259 290x30), "%s", text variable: GVL_RecipeTable.aRecipeNames[GVL_RecipeTable.nRecipeIndex+6], colour toggle: (GVL_RecipeTable.nRecipeSelectionIndex-GVL_RecipeTable.nRecipeIndex) = 6
        OnMouseDown: execute { GVL_RecipeTable.nRecipeSelectionIndex := GVL_RecipeTable.nRecipeIndex + 6; }
    Rectangle (891,289 290x30), "%s", text variable: GVL_RecipeTable.aRecipeNames[GVL_RecipeTable.nRecipeIndex+7], colour toggle: (GVL_RecipeTable.nRecipeSelectionIndex-GVL_RecipeTable.nRecipeIndex) = 7
        OnMouseDown: execute { GVL_RecipeTable.nRecipeSelectionIndex := GVL_RecipeTable.nRecipeIndex + 7; }
    Rectangle (891,319 290x30), "%s", text variable: GVL_RecipeTable.aRecipeNames[GVL_RecipeTable.nRecipeIndex+8], colour toggle: (GVL_RecipeTable.nRecipeSelectionIndex-GVL_RecipeTable.nRecipeIndex) = 8
        OnMouseDown: execute { GVL_RecipeTable.nRecipeSelectionIndex := GVL_RecipeTable.nRecipeIndex + 8; }
    Rectangle (891,349 290x30), "%s", text variable: GVL_RecipeTable.aRecipeNames[GVL_RecipeTable.nRecipeIndex+9], colour toggle: (GVL_RecipeTable.nRecipeSelectionIndex-GVL_RecipeTable.nRecipeIndex) = 9
        OnMouseDown: execute { GVL_RecipeTable.nRecipeSelectionIndex := GVL_RecipeTable.nRecipeIndex + 9; }
    Rectangle (891,379 321x30), "Wybrany numer recepty: %s", text variable: GVL_RecipeTable.nRecipeSelectionIndex+1, input disabled if: TRUE
    Scrollbar (1182,79 30x300)
        p2245068023: GVL_RecipeTable.nRecipeCount
        p1057716461: GVL_RecipeTable.nRecipeIndex
    Group (884,498 321x209)
        Label (0,29 321x31), "1. Naciśnij wolny wiersz w tabeli "Recepty","
        Label (1,0 271x30), "UWAGA !!! TWORZENIE NOWEJ RECEPTY"
        Label (0,59 150x30), "a następnie"Create recipe""
        Label (0,149 150x30), "4. Naciśnij " Save""
        Label (0,89 150x30), "2. Naciśnij " Save as""
        Label (0,179 150x30)
        Label (0,119 183x30), "3. Wprowadź wartości do tabeli"
        Label (0,179 150x30), "5. Naciśnij "Save recipe""
    Button (446,476 350x30), "Value"
    Button (797,476 31x27), "Save"
        OnMouseDown: toggle RecipeManagement.bSaveVariables
    Rectangle (445,506 350x30), "%s", text variable: GVL_RecipeTable.aVariableValues[GVL_RecipeTable.nVariableIndex]
        OnMouseDown: write the text variable via Edit
    Rectangle (445,536 350x30), "%s", text variable: GVL_RecipeTable.aVariableValues[GVL_RecipeTable.nVariableIndex+1]
        OnMouseDown: write the text variable via Edit
    Rectangle (445,566 350x30), "%s", text variable: GVL_RecipeTable.aVariableValues[GVL_RecipeTable.nVariableIndex+2]
        OnMouseDown: write the text variable via Edit
    Rectangle (445,596 350x30), "%s", text variable: GVL_RecipeTable.aVariableValues[GVL_RecipeTable.nVariableIndex+3]
        OnMouseDown: write the text variable via Edit
    Rectangle (445,626 350x30), "%s", text variable: GVL_RecipeTable.aVariableValues[GVL_RecipeTable.nVariableIndex+4]
        OnMouseDown: write the text variable via Edit
    Scrollbar (797,506 29x181)
        p1057716461: GVL_RecipeTable.nVariableIndex
    Rectangle (445,656 350x30), "%s", text variable: GVL_RecipeTable.aVariableValues[GVL_RecipeTable.nVariableIndex+5]
        OnMouseDown: write the text variable via Edit
    Button (45,476 400x30), "Name"
    Textfield (44,506 400x29), "%s", text variable: GVL_RecipeTable.aVariableNames[GVL_RecipeTable.nVariableIndex], input disabled if: TRUE
        OnMouseClick: write the text variable via Default
    Textfield (44,536 400x29), "%s", text variable: GVL_RecipeTable.aVariableNames[GVL_RecipeTable.nVariableIndex+1], input disabled if: TRUE
        OnMouseClick: write the text variable via Default
    Textfield (44,566 400x29), "%s", text variable: GVL_RecipeTable.aVariableNames[GVL_RecipeTable.nVariableIndex+2], input disabled if: TRUE
        OnMouseClick: write the text variable via Default
    Textfield (44,596 400x29), "%s", text variable: GVL_RecipeTable.aVariableNames[GVL_RecipeTable.nVariableIndex+3], input disabled if: TRUE
        OnMouseClick: write the text variable via Default
    Textfield (44,626 400x29), "%s", text variable: GVL_RecipeTable.aVariableNames[GVL_RecipeTable.nVariableIndex+4], input disabled if: TRUE
        OnMouseClick: write the text variable via Default
    Textfield (44,656 400x29), "%s", text variable: GVL_RecipeTable.aVariableNames[GVL_RecipeTable.nVariableIndex+5], input disabled if: TRUE
        OnMouseClick: write the text variable via Default
    Button (446,236 350x30), "Value"
    Rectangle (445,266 350x30), "%s", text variable: GVL_RecipeTable.aCurrentValues[GVL_RecipeTable.nVariableIndex], input disabled if: TRUE
        OnMouseDown: write the text variable via Edit
    Rectangle (445,296 350x30), "%s", text variable: GVL_RecipeTable.aCurrentValues[GVL_RecipeTable.nVariableIndex+1], input disabled if: TRUE
        OnMouseDown: write the text variable via Edit
    Rectangle (445,326 350x30), "%s", text variable: GVL_RecipeTable.aCurrentValues[GVL_RecipeTable.nVariableIndex+2], input disabled if: TRUE
        OnMouseDown: write the text variable via Edit
    Rectangle (445,356 350x30), "%s", text variable: GVL_RecipeTable.aCurrentValues[GVL_RecipeTable.nVariableIndex+3], input disabled if: TRUE
        OnMouseDown: write the text variable via Edit
    Rectangle (445,386 350x30), "%s", text variable: GVL_RecipeTable.aCurrentValues[GVL_RecipeTable.nVariableIndex+4], input disabled if: TRUE
        OnMouseDown: write the text variable via Edit
    Scrollbar (797,236 29x211)
        p1057716461: GVL_RecipeTable.nVariableIndex1
    Rectangle (445,416 350x30), "%s", text variable: GVL_RecipeTable.aCurrentValues[GVL_RecipeTable.nVariableIndex+5], input disabled if: TRUE
        OnMouseDown: write the text variable via Edit
    Button (45,236 400x30), "Name"
    Label (906,427 150x30), "Nazwa Recepty"
    Textfield (1049,427 150x30), "%s", text variable: MAIN.sRecipe
END_VISUALIZATION

// ---- VISUs/Zaklejarka.TcVIS
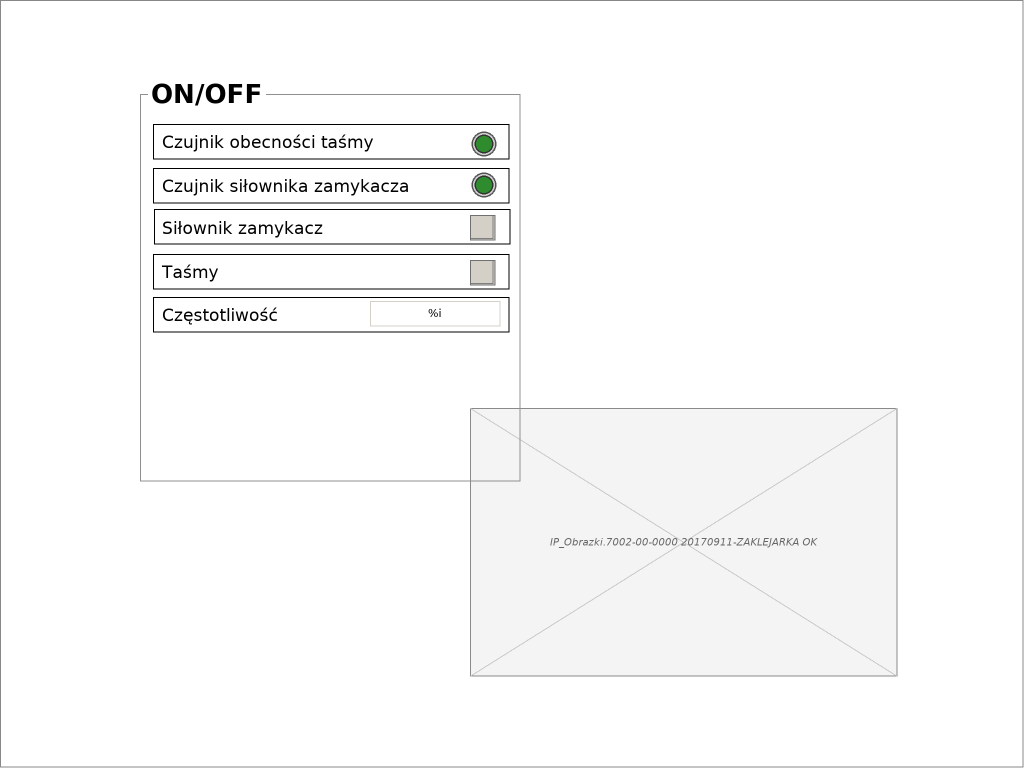
VISUALIZATION Zaklejarka  // 1024x768
    Image (470,408 427x268), image: IP_Obrazki.7002-00-0000 20170911-ZAKLEJARKA OK
    GroupBox (140,86 380x395), "ON/OFF"
        Rectangle (14,123 356x35)
        Rectangle (13,168 356x35)
        Rectangle (13,38 356x35)
        Label (19,41 230x30), "Czujnik obecności taśmy"
        Rectangle (13,82 356x35)
        Label (19,85 239x30), "Czujnik siłownika zamykacza"
        Label (19,171 209x30), "Taśmy"
        Label (19,127 209x30), "Siłownik zamykacz"
        Rectangle (13,211 356x35)
        Lamp1 (330,85 28x28), variable: GVL_Zak_IO.b_kZamykacz1, style: Lamp-Lamp1-Green
        Lamp1 (330,44 28x28), variable: GVL_Zak_IO.b_czujnik_OT, style: Lamp-Lamp1-Green
        Label (19,299 209x30)
        Textfield (230,215 130x25), "%i", text variable: GVL_HMI.iFreqKierownicaMan
            OnMouseClick: write the text variable via Edit
        Button (330,129 25x25), colour toggle: GVL_GLOBAL.zaw_klap_krot_cewka
            tap GVL_HMI.przycisk_sil_zamykacz_zaklejarka
        Button (330,174 25x25), colour toggle: GVL_GLOBAL.tasmy_zaklejarka_cewka
            tap GVL_HMI.przycisk_tasmy_zaklejarka
    Label (159,300 209x30), "Częstotliwość"
END_VISUALIZATION
